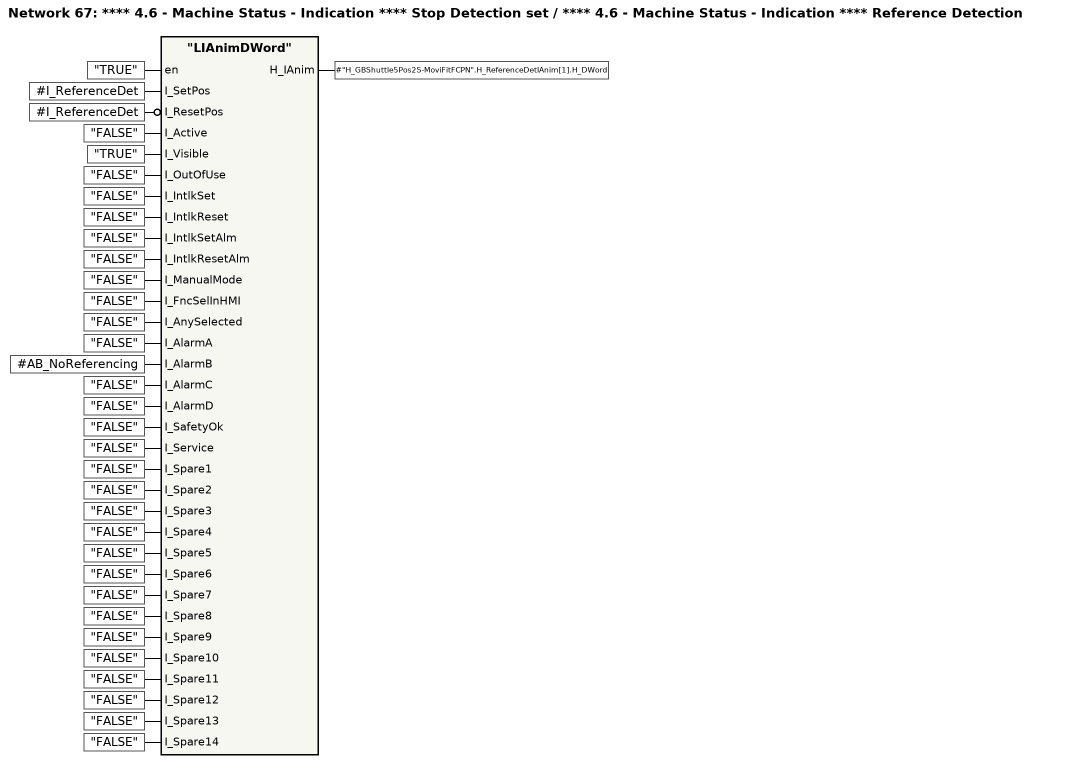
   IF "TRUE" THEN
       "LIAnimDWord"(I_SetPos := #I_ReferenceDet,
                     I_ResetPos := NOT #I_ReferenceDet,
                     I_Active := "FALSE",
                     I_Visible := "TRUE",
                     I_OutOfUse := "FALSE",
                     I_IntlkSet := "FALSE",
                     I_IntlkReset := "FALSE",
                     I_IntlkSetAlm := "FALSE",
                     I_IntlkResetAlm := "FALSE",
                     I_ManualMode := "FALSE",
                     I_FncSelInHMI := "FALSE",
                     I_AnySelected := "FALSE",
                     I_AlarmA := "FALSE",
                     I_AlarmB := #AB_NoReferencing,
                     I_AlarmC := "FALSE",
                     I_AlarmD := "FALSE",
                     I_SafetyOk := "FALSE",
                     I_Service := "FALSE",
                     I_Spare1 := "FALSE",
                     I_Spare2 := "FALSE",
                     I_Spare3 := "FALSE",
                     I_Spare4 := "FALSE",
                     I_Spare5 := "FALSE",
                     I_Spare6 := "FALSE",
                     I_Spare7 := "FALSE",
                     I_Spare8 := "FALSE",
                     I_Spare9 := "FALSE",
                     I_Spare10 := "FALSE",
                     I_Spare11 := "FALSE",
                     I_Spare12 := "FALSE",
                     I_Spare13 := "FALSE",
                     I_Spare14 := "FALSE",
                     H_IAnim => #"H_GBShuttle5Pos2S-MoviFitFCPN".H_ReferenceDetIAnim[1].H_DWord);
   END_IF;
END_REGION

REGION Network 68: **** 4.6 - Machine status - Indications **** Icon Animation
   // Animation for HMI
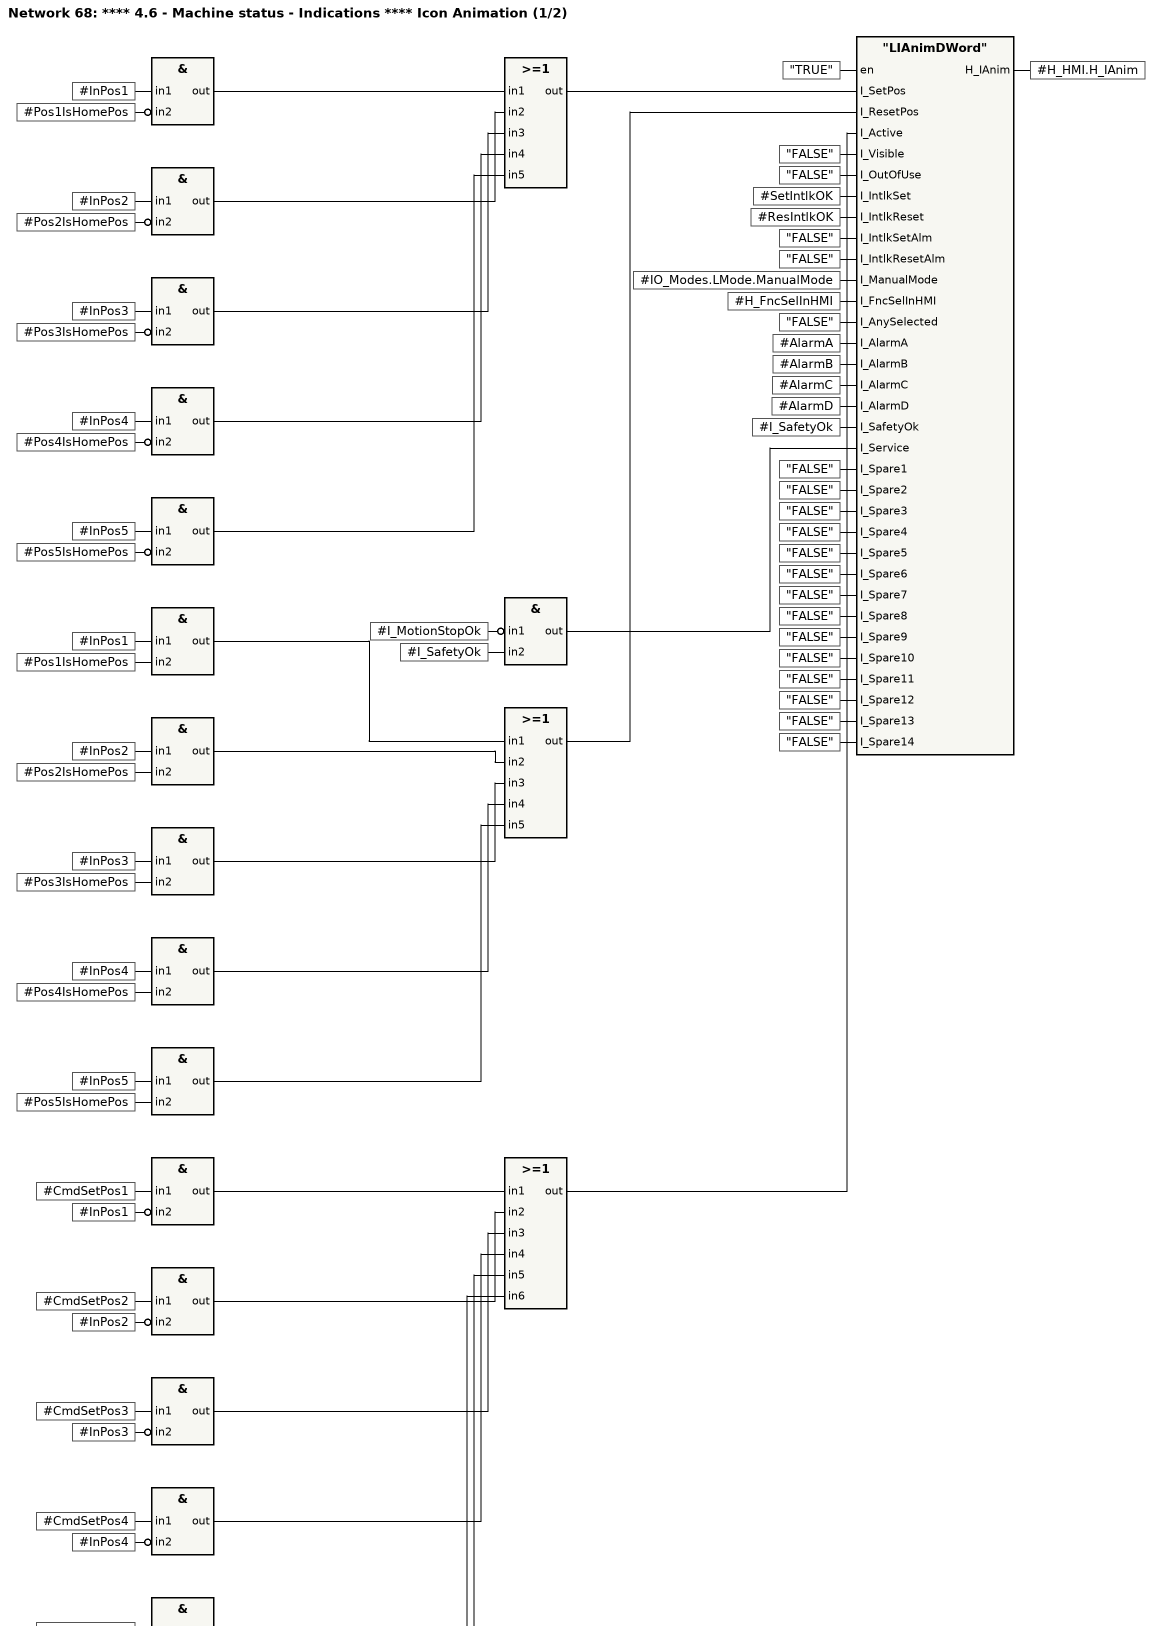
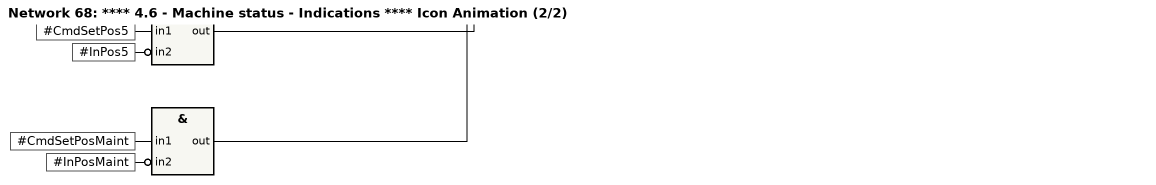
   IF "TRUE" THEN
       "LIAnimDWord"(I_SetPos := (#InPos1 AND NOT #Pos1IsHomePos) OR (#InPos2 AND NOT #Pos2IsHomePos) OR (#InPos3 AND NOT #Pos3IsHomePos) OR (#InPos4 AND NOT #Pos4IsHomePos) OR (#InPos5 AND NOT #Pos5IsHomePos),
                     I_ResetPos := (#InPos1 AND #Pos1IsHomePos) OR (#InPos2 AND #Pos2IsHomePos) OR (#InPos3 AND #Pos3IsHomePos) OR (#InPos4 AND #Pos4IsHomePos) OR (#InPos5 AND #Pos5IsHomePos),
                     I_Active := (#CmdSetPos1 AND NOT #InPos1) OR (#CmdSetPos2 AND NOT #InPos2) OR (#CmdSetPos3 AND NOT #InPos3) OR (#CmdSetPos4 AND NOT #InPos4) OR (#CmdSetPos5 AND NOT #InPos5) OR (#CmdSetPosMaint AND NOT #InPosMaint),
                     I_Visible := "FALSE",
                     I_OutOfUse := "FALSE",
                     I_IntlkSet := #SetIntlkOK,
                     I_IntlkReset := #ResIntlkOK,
                     I_IntlkSetAlm := "FALSE",
                     I_IntlkResetAlm := "FALSE",
                     I_ManualMode := #IO_Modes.LMode.ManualMode,
                     I_FncSelInHMI := #H_FncSelInHMI,
                     I_AnySelected := "FALSE",
                     I_AlarmA := #AlarmA,
                     I_AlarmB := #AlarmB,
                     I_AlarmC := #AlarmC,
                     I_AlarmD := #AlarmD,
                     I_SafetyOk := #I_SafetyOk,
                     I_Service := NOT #I_MotionStopOk AND #I_SafetyOk,
                     I_Spare1 := "FALSE",
                     I_Spare2 := "FALSE",
                     I_Spare3 := "FALSE",
                     I_Spare4 := "FALSE",
                     I_Spare5 := "FALSE",
                     I_Spare6 := "FALSE",
                     I_Spare7 := "FALSE",
                     I_Spare8 := "FALSE",
                     I_Spare9 := "FALSE",
                     I_Spare10 := "FALSE",
                     I_Spare11 := "FALSE",
                     I_Spare12 := "FALSE",
                     I_Spare13 := "FALSE",
                     I_Spare14 := "FALSE",
                     H_IAnim => #H_HMI.H_IAnim);
   END_IF;
END_REGION

REGION Network 69: **** 4.6 - Machine status - Indications **** Anim / **** 4.6 - Machine status - Indications **** Animation
   // Animation for HMI
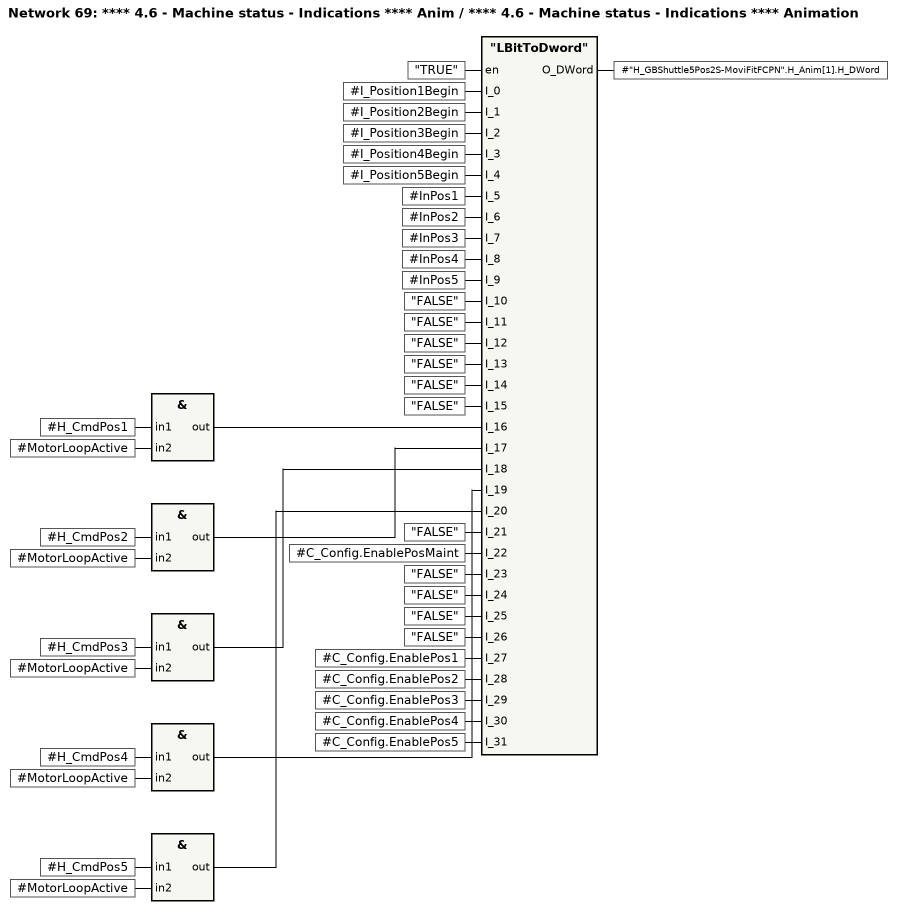
   IF "TRUE" THEN
       "LBitToDword"(I_0 := #I_Position1Begin,
                     I_1 := #I_Position2Begin,
                     I_2 := #I_Position3Begin,
                     I_3 := #I_Position4Begin,
                     I_4 := #I_Position5Begin,
                     I_5 := #InPos1,
                     I_6 := #InPos2,
                     I_7 := #InPos3,
                     I_8 := #InPos4,
                     I_9 := #InPos5,
                     I_10 := "FALSE",
                     I_11 := "FALSE",
                     I_12 := "FALSE",
                     I_13 := "FALSE",
                     I_14 := "FALSE",
                     I_15 := "FALSE",
                     I_16 := #H_CmdPos1 AND #MotorLoopActive,
                     I_17 := #H_CmdPos2 AND #MotorLoopActive,
                     I_18 := #H_CmdPos3 AND #MotorLoopActive,
                     I_19 := #H_CmdPos4 AND #MotorLoopActive,
                     I_20 := #H_CmdPos5 AND #MotorLoopActive,
                     I_21 := "FALSE",
                     I_22 := #C_Config.EnablePosMaint,
                     I_23 := "FALSE",
                     I_24 := "FALSE",
                     I_25 := "FALSE",
                     I_26 := "FALSE",
                     I_27 := #C_Config.EnablePos1,
                     I_28 := #C_Config.EnablePos2,
                     I_29 := #C_Config.EnablePos3,
                     I_30 := #C_Config.EnablePos4,
                     I_31 := #C_Config.EnablePos5,
                     O_DWord => #"H_GBShuttle5Pos2S-MoviFitFCPN".H_Anim[1].H_DWord);
   END_IF;
END_REGION

REGION Network 70: **** 4.6 - Machine status - Indications **** Anim / **** 4.6 - Machine status - Indications **** Animation
   // Animation for HMI
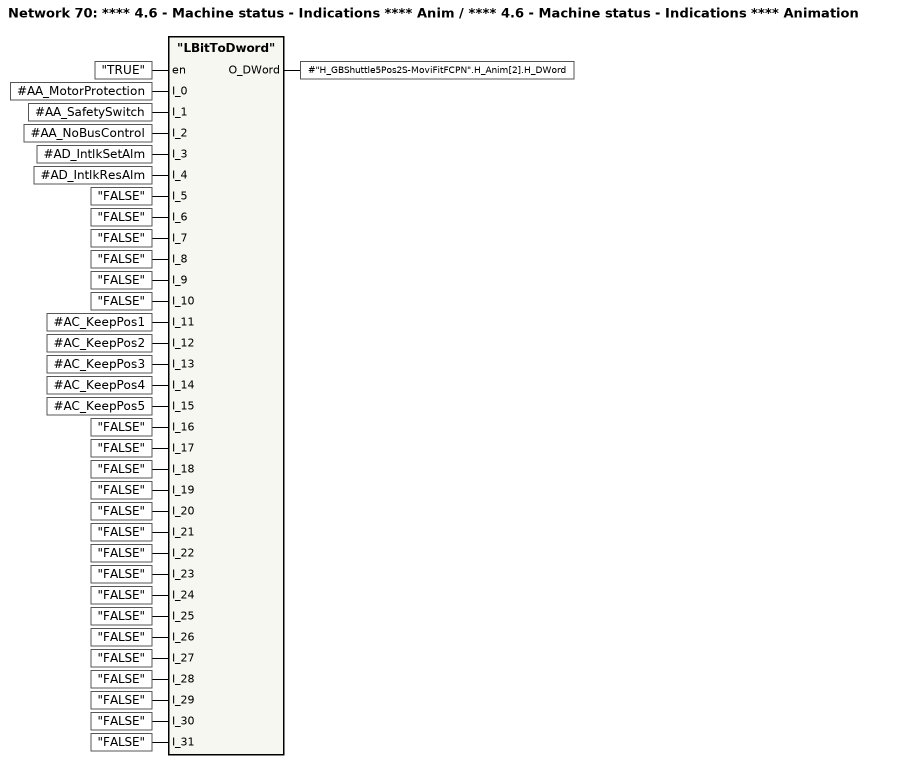
   IF "TRUE" THEN
       "LBitToDword"(I_0 := #AA_MotorProtection,
                     I_1 := #AA_SafetySwitch,
                     I_2 := #AA_NoBusControl,
                     I_3 := #AD_IntlkSetAlm,
                     I_4 := #AD_IntlkResAlm,
                     I_5 := "FALSE",
                     I_6 := "FALSE",
                     I_7 := "FALSE",
                     I_8 := "FALSE",
                     I_9 := "FALSE",
                     I_10 := "FALSE",
                     I_11 := #AC_KeepPos1,
                     I_12 := #AC_KeepPos2,
                     I_13 := #AC_KeepPos3,
                     I_14 := #AC_KeepPos4,
                     I_15 := #AC_KeepPos5,
                     I_16 := "FALSE",
                     I_17 := "FALSE",
                     I_18 := "FALSE",
                     I_19 := "FALSE",
                     I_20 := "FALSE",
                     I_21 := "FALSE",
                     I_22 := "FALSE",
                     I_23 := "FALSE",
                     I_24 := "FALSE",
                     I_25 := "FALSE",
                     I_26 := "FALSE",
                     I_27 := "FALSE",
                     I_28 := "FALSE",
                     I_29 := "FALSE",
                     I_30 := "FALSE",
                     I_31 := "FALSE",
                     O_DWord => #"H_GBShuttle5Pos2S-MoviFitFCPN".H_Anim[2].H_DWord);
   END_IF;
END_REGION

REGION Network 71: **** 4.6 - Machine status - Indications **** Anim / **** 4.6 - Machine status - Indications **** Animation
   // Animation for HMI
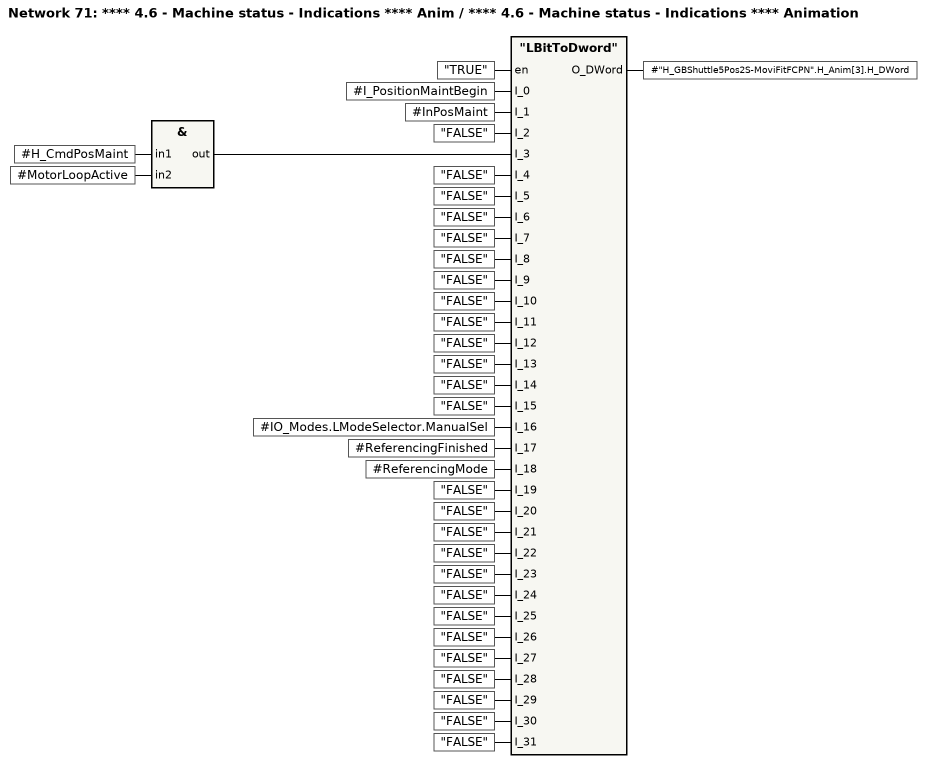
   IF "TRUE" THEN
       "LBitToDword"(I_0 := #I_PositionMaintBegin,
                     I_1 := #InPosMaint,
                     I_2 := "FALSE",
                     I_3 := #H_CmdPosMaint AND #MotorLoopActive,
                     I_4 := "FALSE",
                     I_5 := "FALSE",
                     I_6 := "FALSE",
                     I_7 := "FALSE",
                     I_8 := "FALSE",
                     I_9 := "FALSE",
                     I_10 := "FALSE",
                     I_11 := "FALSE",
                     I_12 := "FALSE",
                     I_13 := "FALSE",
                     I_14 := "FALSE",
                     I_15 := "FALSE",
                     I_16 := #IO_Modes.LModeSelector.ManualSel,
                     I_17 := #ReferencingFinished,
                     I_18 := #ReferencingMode,
                     I_19 := "FALSE",
                     I_20 := "FALSE",
                     I_21 := "FALSE",
                     I_22 := "FALSE",
                     I_23 := "FALSE",
                     I_24 := "FALSE",
                     I_25 := "FALSE",
                     I_26 := "FALSE",
                     I_27 := "FALSE",
                     I_28 := "FALSE",
                     I_29 := "FALSE",
                     I_30 := "FALSE",
                     I_31 := "FALSE",
                     O_DWord => #"H_GBShuttle5Pos2S-MoviFitFCPN".H_Anim[3].H_DWord);
   END_IF;
END_REGION

REGION Network 72: **** 4.6 - Machine status - Indications **** Anim / **** 4.6 - Machine status - Indications **** Animation
   // Anim
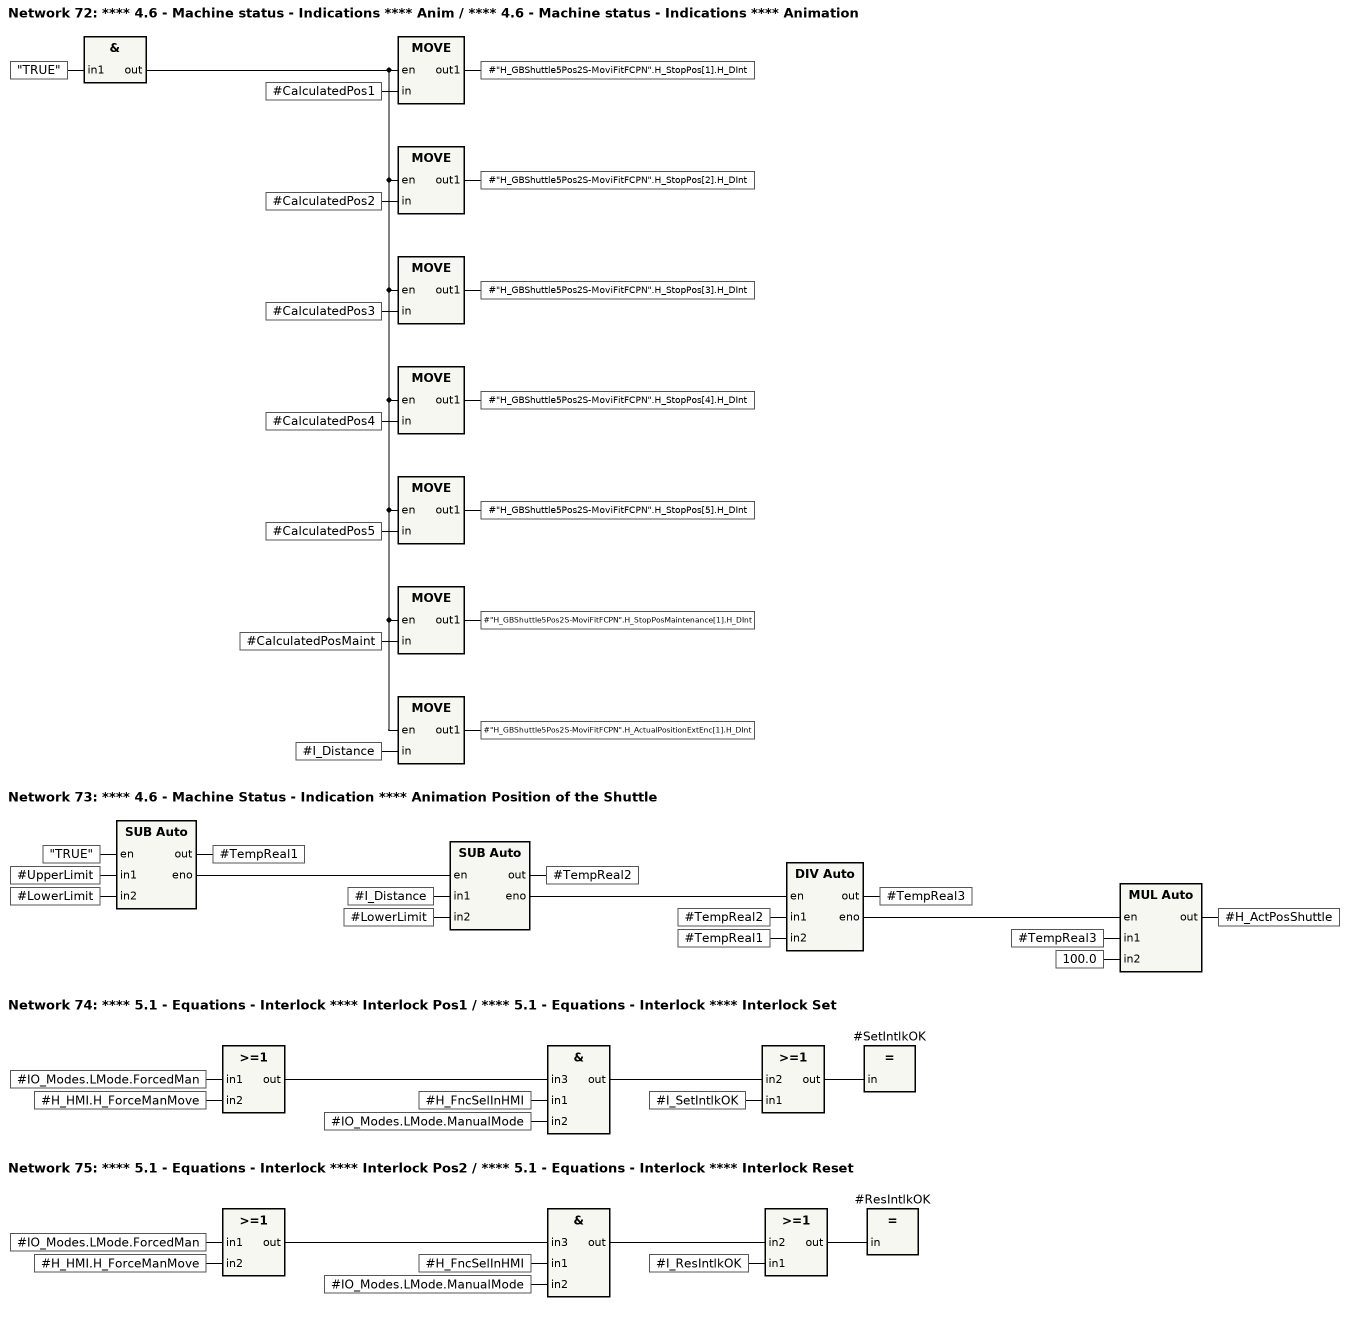
   IF "TRUE" THEN
       #"H_GBShuttle5Pos2S-MoviFitFCPN".H_StopPos[1].H_DInt := #CalculatedPos1;
       #"H_GBShuttle5Pos2S-MoviFitFCPN".H_StopPos[2].H_DInt := #CalculatedPos2;
       #"H_GBShuttle5Pos2S-MoviFitFCPN".H_StopPos[3].H_DInt := #CalculatedPos3;
       #"H_GBShuttle5Pos2S-MoviFitFCPN".H_StopPos[4].H_DInt := #CalculatedPos4;
       #"H_GBShuttle5Pos2S-MoviFitFCPN".H_StopPos[5].H_DInt := #CalculatedPos5;
       #"H_GBShuttle5Pos2S-MoviFitFCPN".H_StopPosMaintenance[1].H_DInt := #CalculatedPosMaint;
       #"H_GBShuttle5Pos2S-MoviFitFCPN".H_ActualPositionExtEnc[1].H_DInt := #I_Distance;
   END_IF;
END_REGION

REGION Network 73: **** 4.6 - Machine Status - Indication **** Animation Position of the Shuttle
   IF "TRUE" THEN
       #TempReal1 := #UpperLimit - #LowerLimit;
       #TempReal2 := #I_Distance - #LowerLimit;
       #TempReal3 := #TempReal2 / #TempReal1;
       #H_ActPosShuttle := #TempReal3 * 100.0;
   END_IF;
END_REGION

REGION Network 74: **** 5.1 - Equations - Interlock **** Interlock Pos1 / **** 5.1 - Equations - Interlock **** Interlock Set
   // Interlock
   #SetIntlkOK := ((#IO_Modes.LMode.ForcedMan OR #H_HMI.H_ForceManMove) AND #H_FncSelInHMI AND #IO_Modes.LMode.ManualMode) OR #I_SetIntlkOK;
END_REGION

REGION Network 75: **** 5.1 - Equations - Interlock **** Interlock Pos2 / **** 5.1 - Equations - Interlock **** Interlock Reset
   // Interlock
   #ResIntlkOK := ((#IO_Modes.LMode.ForcedMan OR #H_HMI.H_ForceManMove) AND #H_FncSelInHMI AND #IO_Modes.LMode.ManualMode) OR #I_ResIntlkOK;
END_REGION

REGION Network 76: **** 5.2 - Equations - Equations **** Alarm Condition Keep Position 1
   // Alarm Condition Keep Position
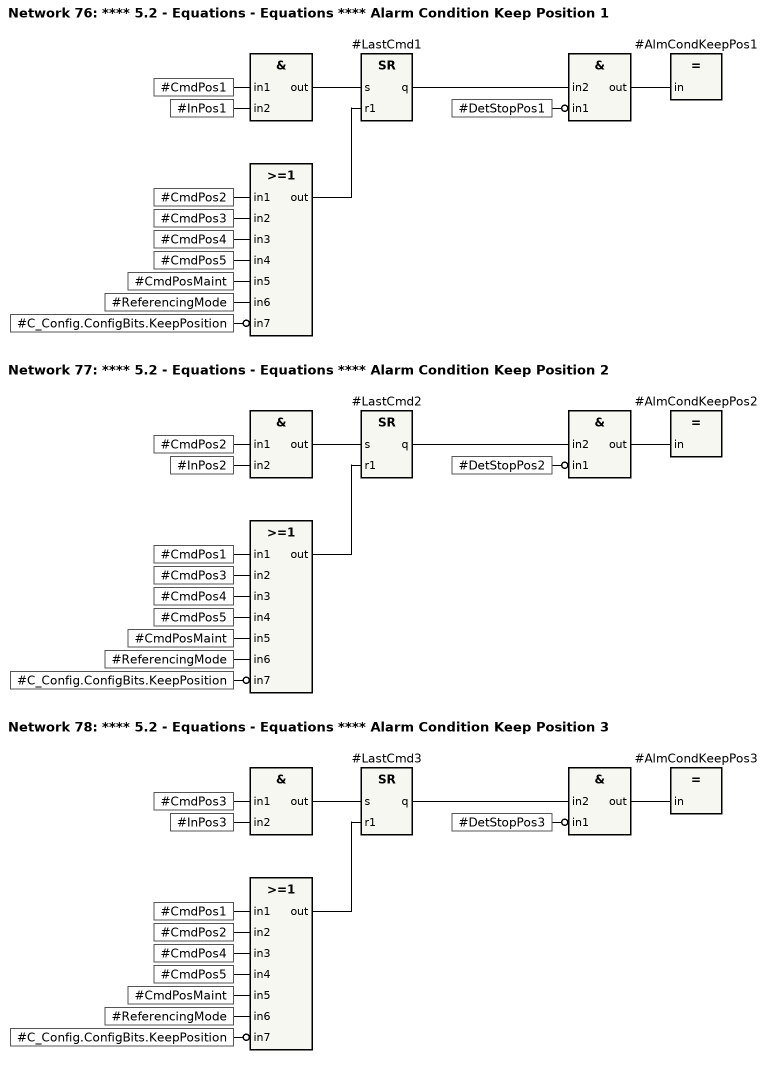
   IF #CmdPos1 AND #InPos1 THEN
       #LastCmd1 := TRUE;   // SR flip-flop
   END_IF;
   IF #CmdPos2 OR #CmdPos3 OR #CmdPos4 OR #CmdPos5 OR #CmdPosMaint OR #ReferencingMode OR NOT #C_Config.ConfigBits.KeepPosition THEN
       #LastCmd1 := FALSE;
   END_IF;
   #AlmCondKeepPos1 := #LastCmd1 AND NOT #DetStopPos1;
END_REGION

REGION Network 77: **** 5.2 - Equations - Equations **** Alarm Condition Keep Position 2
   // Alarm Condition Keep Position
   IF #CmdPos2 AND #InPos2 THEN
       #LastCmd2 := TRUE;   // SR flip-flop
   END_IF;
   IF #CmdPos1 OR #CmdPos3 OR #CmdPos4 OR #CmdPos5 OR #CmdPosMaint OR #ReferencingMode OR NOT #C_Config.ConfigBits.KeepPosition THEN
       #LastCmd2 := FALSE;
   END_IF;
   #AlmCondKeepPos2 := #LastCmd2 AND NOT #DetStopPos2;
END_REGION

REGION Network 78: **** 5.2 - Equations - Equations **** Alarm Condition Keep Position 3
   // Alarm Condition Keep Position
   IF #CmdPos3 AND #InPos3 THEN
       #LastCmd3 := TRUE;   // SR flip-flop
   END_IF;
   IF #CmdPos1 OR #CmdPos2 OR #CmdPos4 OR #CmdPos5 OR #CmdPosMaint OR #ReferencingMode OR NOT #C_Config.ConfigBits.KeepPosition THEN
       #LastCmd3 := FALSE;
   END_IF;
   #AlmCondKeepPos3 := #LastCmd3 AND NOT #DetStopPos3;
END_REGION

REGION Network 79: **** 5.2 - Equations - Equations **** Alarm Condition Keep Position 4
   // Alarm Condition Keep Position
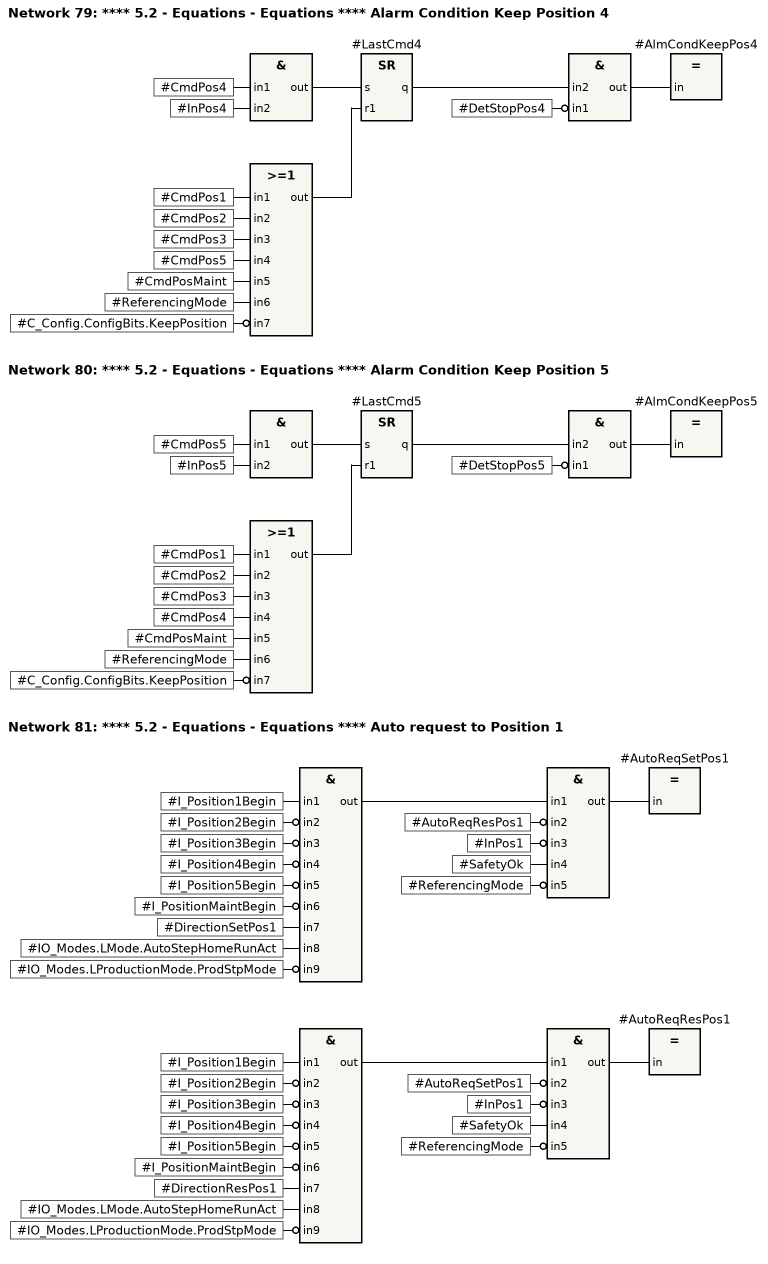
   IF #CmdPos4 AND #InPos4 THEN
       #LastCmd4 := TRUE;   // SR flip-flop
   END_IF;
   IF #CmdPos1 OR #CmdPos2 OR #CmdPos3 OR #CmdPos5 OR #CmdPosMaint OR #ReferencingMode OR NOT #C_Config.ConfigBits.KeepPosition THEN
       #LastCmd4 := FALSE;
   END_IF;
   #AlmCondKeepPos4 := #LastCmd4 AND NOT #DetStopPos4;
END_REGION

REGION Network 80: **** 5.2 - Equations - Equations **** Alarm Condition Keep Position 5
   // Alarm Condition Keep Position
   IF #CmdPos5 AND #InPos5 THEN
       #LastCmd5 := TRUE;   // SR flip-flop
   END_IF;
   IF #CmdPos1 OR #CmdPos2 OR #CmdPos3 OR #CmdPos4 OR #CmdPosMaint OR #ReferencingMode OR NOT #C_Config.ConfigBits.KeepPosition THEN
       #LastCmd5 := FALSE;
   END_IF;
   #AlmCondKeepPos5 := #LastCmd5 AND NOT #DetStopPos5;
END_REGION

REGION Network 81: **** 5.2 - Equations - Equations **** Auto request to Position 1
   // AutoReq Pos 1
   #AutoReqSetPos1 := #I_Position1Begin AND NOT #I_Position2Begin AND NOT #I_Position3Begin AND NOT #I_Position4Begin AND NOT #I_Position5Begin AND NOT #I_PositionMaintBegin AND #DirectionSetPos1 AND #IO_Modes.LMode.AutoStepHomeRunAct AND NOT #IO_Modes.LProductionMode.ProdStpMode AND NOT #AutoReqResPos1 AND NOT #InPos1 AND #SafetyOk AND NOT #ReferencingMode;
   #AutoReqResPos1 := #I_Position1Begin AND NOT #I_Position2Begin AND NOT #I_Position3Begin AND NOT #I_Position4Begin AND NOT #I_Position5Begin AND NOT #I_PositionMaintBegin AND #DirectionResPos1 AND #IO_Modes.LMode.AutoStepHomeRunAct AND NOT #IO_Modes.LProductionMode.ProdStpMode AND NOT #AutoReqSetPos1 AND NOT #InPos1 AND #SafetyOk AND NOT #ReferencingMode;
END_REGION

REGION Network 82: **** 5.2 - Equations - Equations **** Auto request to Position 2
   // AutoReq Pos 1
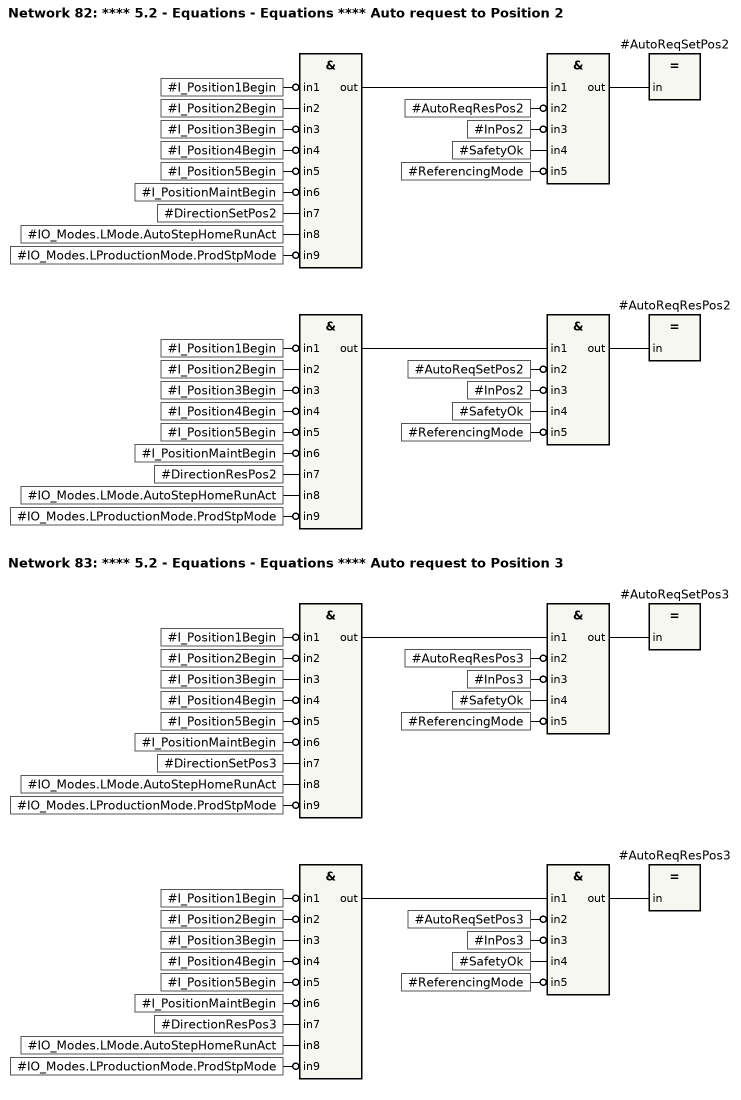
   #AutoReqSetPos2 := NOT #I_Position1Begin AND #I_Position2Begin AND NOT #I_Position3Begin AND NOT #I_Position4Begin AND NOT #I_Position5Begin AND NOT #I_PositionMaintBegin AND #DirectionSetPos2 AND #IO_Modes.LMode.AutoStepHomeRunAct AND NOT #IO_Modes.LProductionMode.ProdStpMode AND NOT #AutoReqResPos2 AND NOT #InPos2 AND #SafetyOk AND NOT #ReferencingMode;
   #AutoReqResPos2 := NOT #I_Position1Begin AND #I_Position2Begin AND NOT #I_Position3Begin AND NOT #I_Position4Begin AND NOT #I_Position5Begin AND NOT #I_PositionMaintBegin AND #DirectionResPos2 AND #IO_Modes.LMode.AutoStepHomeRunAct AND NOT #IO_Modes.LProductionMode.ProdStpMode AND NOT #AutoReqSetPos2 AND NOT #InPos2 AND #SafetyOk AND NOT #ReferencingMode;
END_REGION

REGION Network 83: **** 5.2 - Equations - Equations **** Auto request to Position 3
   // AutoReq Pos 1
   #AutoReqSetPos3 := NOT #I_Position1Begin AND NOT #I_Position2Begin AND #I_Position3Begin AND NOT #I_Position4Begin AND NOT #I_Position5Begin AND NOT #I_PositionMaintBegin AND #DirectionSetPos3 AND #IO_Modes.LMode.AutoStepHomeRunAct AND NOT #IO_Modes.LProductionMode.ProdStpMode AND NOT #AutoReqResPos3 AND NOT #InPos3 AND #SafetyOk AND NOT #ReferencingMode;
   #AutoReqResPos3 := NOT #I_Position1Begin AND NOT #I_Position2Begin AND #I_Position3Begin AND NOT #I_Position4Begin AND NOT #I_Position5Begin AND NOT #I_PositionMaintBegin AND #DirectionResPos3 AND #IO_Modes.LMode.AutoStepHomeRunAct AND NOT #IO_Modes.LProductionMode.ProdStpMode AND NOT #AutoReqSetPos3 AND NOT #InPos3 AND #SafetyOk AND NOT #ReferencingMode;
END_REGION

REGION Network 84: **** 5.2 - Equations - Equations **** Auto request to Position 4
   // AutoReq Pos 1
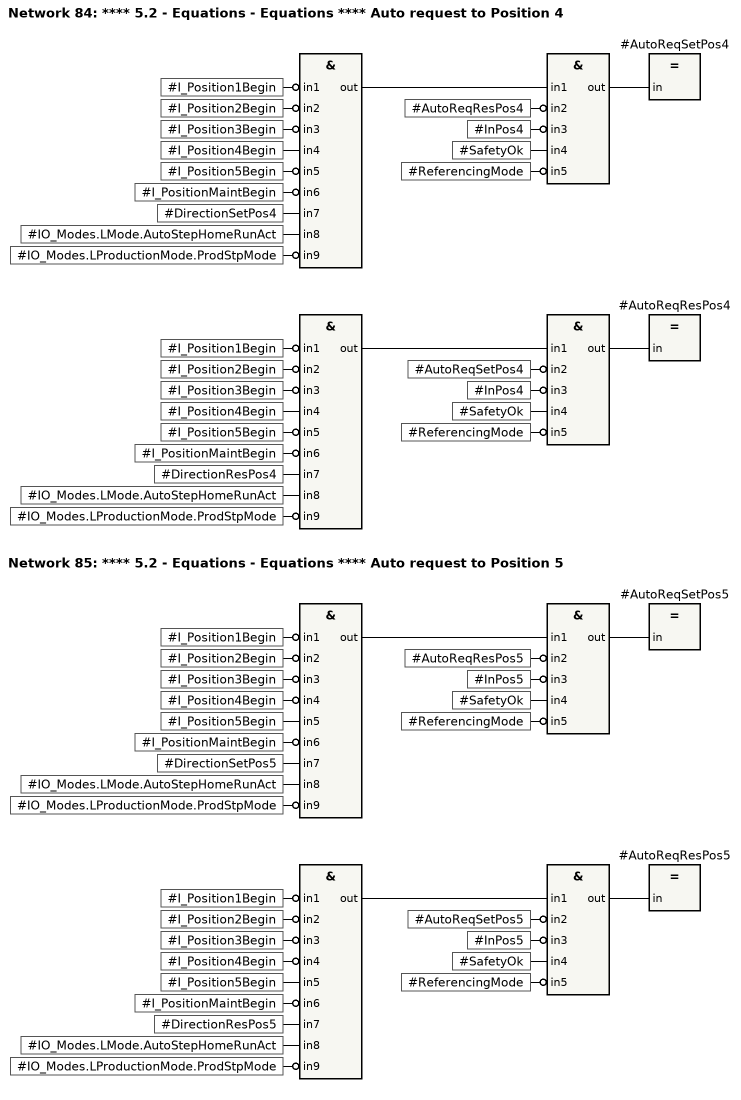
   #AutoReqSetPos4 := NOT #I_Position1Begin AND NOT #I_Position2Begin AND NOT #I_Position3Begin AND #I_Position4Begin AND NOT #I_Position5Begin AND NOT #I_PositionMaintBegin AND #DirectionSetPos4 AND #IO_Modes.LMode.AutoStepHomeRunAct AND NOT #IO_Modes.LProductionMode.ProdStpMode AND NOT #AutoReqResPos4 AND NOT #InPos4 AND #SafetyOk AND NOT #ReferencingMode;
   #AutoReqResPos4 := NOT #I_Position1Begin AND NOT #I_Position2Begin AND NOT #I_Position3Begin AND #I_Position4Begin AND NOT #I_Position5Begin AND NOT #I_PositionMaintBegin AND #DirectionResPos4 AND #IO_Modes.LMode.AutoStepHomeRunAct AND NOT #IO_Modes.LProductionMode.ProdStpMode AND NOT #AutoReqSetPos4 AND NOT #InPos4 AND #SafetyOk AND NOT #ReferencingMode;
END_REGION

REGION Network 85: **** 5.2 - Equations - Equations **** Auto request to Position 5
   // AutoReq Pos 1
   #AutoReqSetPos5 := NOT #I_Position1Begin AND NOT #I_Position2Begin AND NOT #I_Position3Begin AND NOT #I_Position4Begin AND #I_Position5Begin AND NOT #I_PositionMaintBegin AND #DirectionSetPos5 AND #IO_Modes.LMode.AutoStepHomeRunAct AND NOT #IO_Modes.LProductionMode.ProdStpMode AND NOT #AutoReqResPos5 AND NOT #InPos5 AND #SafetyOk AND NOT #ReferencingMode;
   #AutoReqResPos5 := NOT #I_Position1Begin AND NOT #I_Position2Begin AND NOT #I_Position3Begin AND NOT #I_Position4Begin AND #I_Position5Begin AND NOT #I_PositionMaintBegin AND #DirectionResPos5 AND #IO_Modes.LMode.AutoStepHomeRunAct AND NOT #IO_Modes.LProductionMode.ProdStpMode AND NOT #AutoReqSetPos5 AND NOT #InPos5 AND #SafetyOk AND NOT #ReferencingMode;
END_REGION

REGION Network 86: **** 5.2 - Equations - Equations **** Auto request to Position Maintenance
   // AutoReq Pos 1
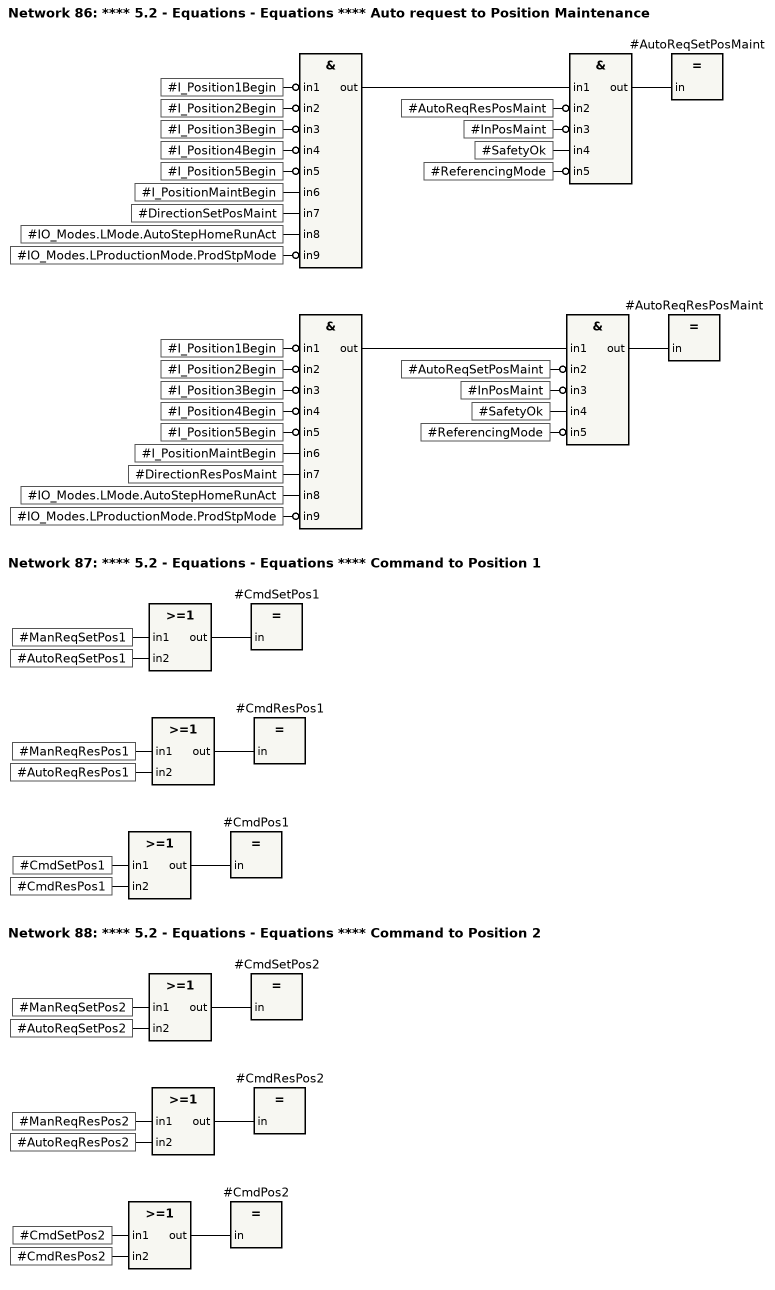
   #AutoReqSetPosMaint := NOT #I_Position1Begin AND NOT #I_Position2Begin AND NOT #I_Position3Begin AND NOT #I_Position4Begin AND NOT #I_Position5Begin AND #I_PositionMaintBegin AND #DirectionSetPosMaint AND #IO_Modes.LMode.AutoStepHomeRunAct AND NOT #IO_Modes.LProductionMode.ProdStpMode AND NOT #AutoReqResPosMaint AND NOT #InPosMaint AND #SafetyOk AND NOT #ReferencingMode;
   #AutoReqResPosMaint := NOT #I_Position1Begin AND NOT #I_Position2Begin AND NOT #I_Position3Begin AND NOT #I_Position4Begin AND NOT #I_Position5Begin AND #I_PositionMaintBegin AND #DirectionResPosMaint AND #IO_Modes.LMode.AutoStepHomeRunAct AND NOT #IO_Modes.LProductionMode.ProdStpMode AND NOT #AutoReqSetPosMaint AND NOT #InPosMaint AND #SafetyOk AND NOT #ReferencingMode;
END_REGION

REGION Network 87: **** 5.2 - Equations - Equations **** Command to Position 1
   #CmdSetPos1 := #ManReqSetPos1 OR #AutoReqSetPos1;
   #CmdResPos1 := #ManReqResPos1 OR #AutoReqResPos1;
   #CmdPos1 := #CmdSetPos1 OR #CmdResPos1;
END_REGION

REGION Network 88: **** 5.2 - Equations - Equations **** Command to Position 2
   #CmdSetPos2 := #ManReqSetPos2 OR #AutoReqSetPos2;
   #CmdResPos2 := #ManReqResPos2 OR #AutoReqResPos2;
   #CmdPos2 := #CmdSetPos2 OR #CmdResPos2;
END_REGION

REGION Network 89: **** 5.2 - Equations - Equations **** Command to Position 3
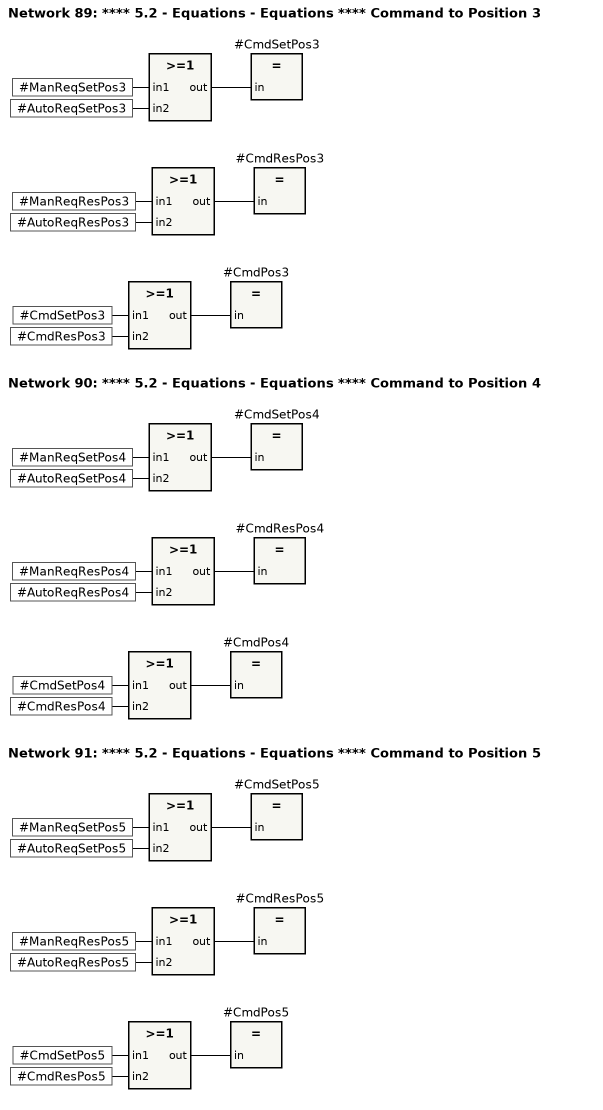
   #CmdSetPos3 := #ManReqSetPos3 OR #AutoReqSetPos3;
   #CmdResPos3 := #ManReqResPos3 OR #AutoReqResPos3;
   #CmdPos3 := #CmdSetPos3 OR #CmdResPos3;
END_REGION

REGION Network 90: **** 5.2 - Equations - Equations **** Command to Position 4
   #CmdSetPos4 := #ManReqSetPos4 OR #AutoReqSetPos4;
   #CmdResPos4 := #ManReqResPos4 OR #AutoReqResPos4;
   #CmdPos4 := #CmdSetPos4 OR #CmdResPos4;
END_REGION

REGION Network 91: **** 5.2 - Equations - Equations **** Command to Position 5
   #CmdSetPos5 := #ManReqSetPos5 OR #AutoReqSetPos5;
   #CmdResPos5 := #ManReqResPos5 OR #AutoReqResPos5;
   #CmdPos5 := #CmdSetPos5 OR #CmdResPos5;
END_REGION

REGION Network 92: **** 5.2 - Equations - Equations **** Command to Position Maintenance
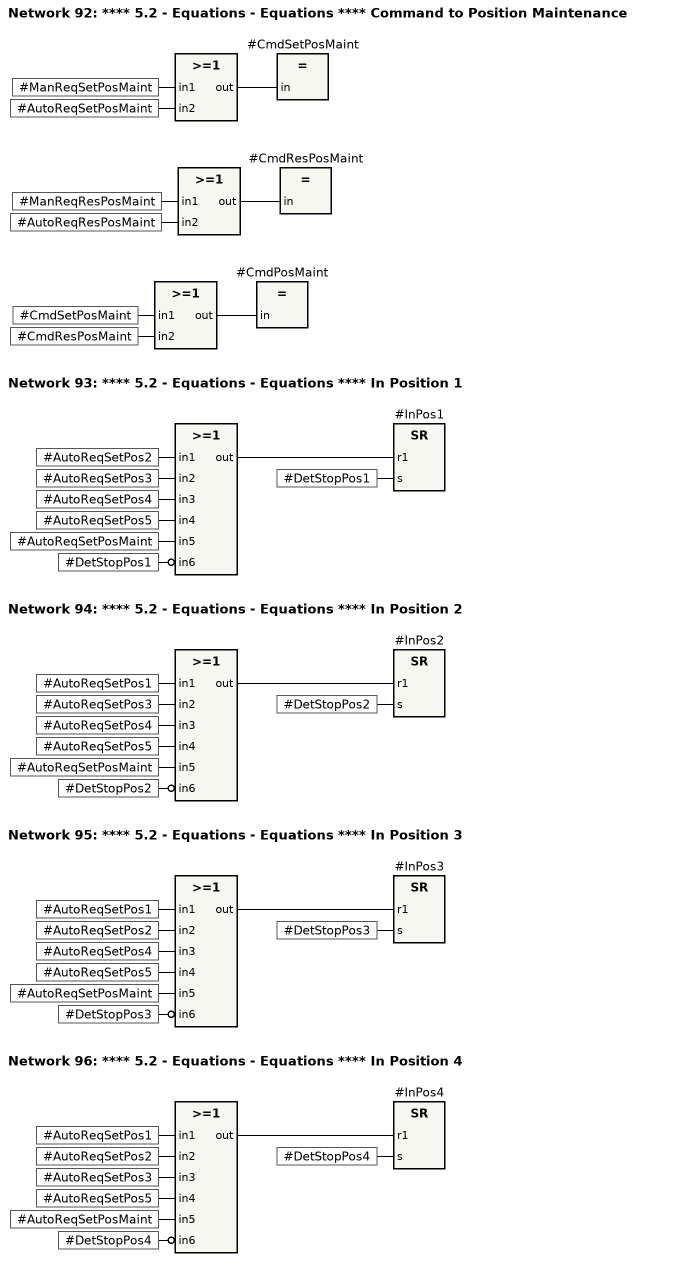
   #CmdSetPosMaint := #ManReqSetPosMaint OR #AutoReqSetPosMaint;
   #CmdResPosMaint := #ManReqResPosMaint OR #AutoReqResPosMaint;
   #CmdPosMaint := #CmdSetPosMaint OR #CmdResPosMaint;
END_REGION

REGION Network 93: **** 5.2 - Equations - Equations **** In Position 1
   IF #DetStopPos1 THEN
       #InPos1 := TRUE;   // SR flip-flop
   END_IF;
   IF #AutoReqSetPos2 OR #AutoReqSetPos3 OR #AutoReqSetPos4 OR #AutoReqSetPos5 OR #AutoReqSetPosMaint OR NOT #DetStopPos1 THEN
       #InPos1 := FALSE;
   END_IF;
END_REGION

REGION Network 94: **** 5.2 - Equations - Equations **** In Position 2
   IF #DetStopPos2 THEN
       #InPos2 := TRUE;   // SR flip-flop
   END_IF;
   IF #AutoReqSetPos1 OR #AutoReqSetPos3 OR #AutoReqSetPos4 OR #AutoReqSetPos5 OR #AutoReqSetPosMaint OR NOT #DetStopPos2 THEN
       #InPos2 := FALSE;
   END_IF;
END_REGION

REGION Network 95: **** 5.2 - Equations - Equations **** In Position 3
   IF #DetStopPos3 THEN
       #InPos3 := TRUE;   // SR flip-flop
   END_IF;
   IF #AutoReqSetPos1 OR #AutoReqSetPos2 OR #AutoReqSetPos4 OR #AutoReqSetPos5 OR #AutoReqSetPosMaint OR NOT #DetStopPos3 THEN
       #InPos3 := FALSE;
   END_IF;
END_REGION

REGION Network 96: **** 5.2 - Equations - Equations **** In Position 4
   IF #DetStopPos4 THEN
       #InPos4 := TRUE;   // SR flip-flop
   END_IF;
   IF #AutoReqSetPos1 OR #AutoReqSetPos2 OR #AutoReqSetPos3 OR #AutoReqSetPos5 OR #AutoReqSetPosMaint OR NOT #DetStopPos4 THEN
       #InPos4 := FALSE;
   END_IF;
END_REGION

REGION Network 97: **** 5.2 - Equations - Equations **** In Position 5
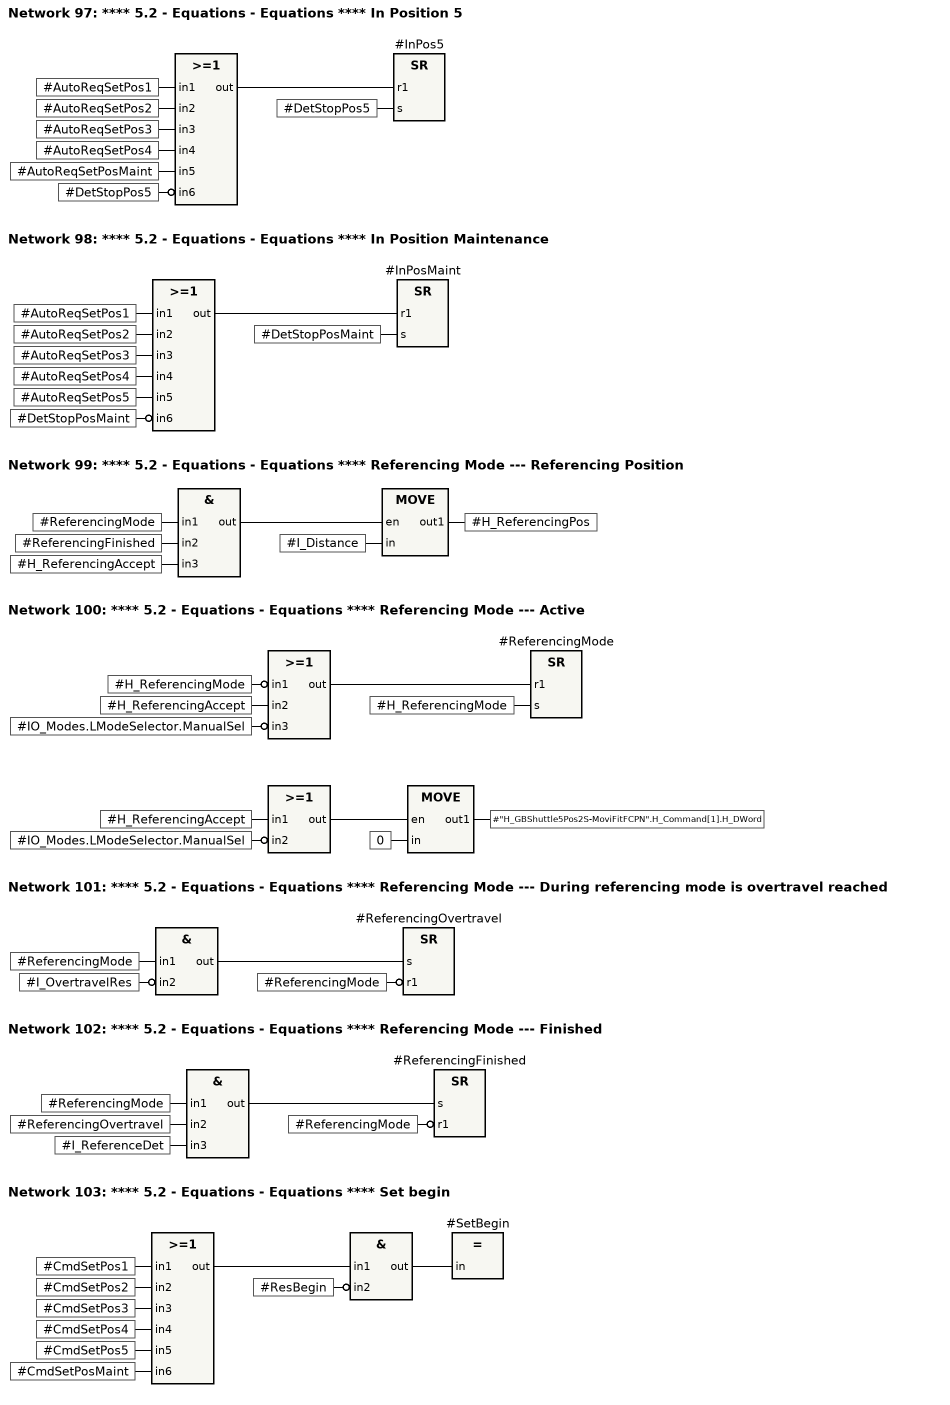
   IF #DetStopPos5 THEN
       #InPos5 := TRUE;   // SR flip-flop
   END_IF;
   IF #AutoReqSetPos1 OR #AutoReqSetPos2 OR #AutoReqSetPos3 OR #AutoReqSetPos4 OR #AutoReqSetPosMaint OR NOT #DetStopPos5 THEN
       #InPos5 := FALSE;
   END_IF;
END_REGION

REGION Network 98: **** 5.2 - Equations - Equations **** In Position Maintenance
   IF #DetStopPosMaint THEN
       #InPosMaint := TRUE;   // SR flip-flop
   END_IF;
   IF #AutoReqSetPos1 OR #AutoReqSetPos2 OR #AutoReqSetPos3 OR #AutoReqSetPos4 OR #AutoReqSetPos5 OR NOT #DetStopPosMaint THEN
       #InPosMaint := FALSE;
   END_IF;
END_REGION

REGION Network 99: **** 5.2 - Equations - Equations **** Referencing Mode --- Referencing Position
   IF #ReferencingMode AND #ReferencingFinished AND #H_ReferencingAccept THEN
       #H_ReferencingPos := #I_Distance;
   END_IF;
END_REGION

REGION Network 100: **** 5.2 - Equations - Equations **** Referencing Mode --- Active
   IF #H_ReferencingMode THEN
       #ReferencingMode := TRUE;   // SR flip-flop
   END_IF;
   IF NOT #H_ReferencingMode OR #H_ReferencingAccept OR NOT #IO_Modes.LModeSelector.ManualSel THEN
       #ReferencingMode := FALSE;
   END_IF;
   IF #H_ReferencingAccept OR NOT #IO_Modes.LModeSelector.ManualSel THEN
       #"H_GBShuttle5Pos2S-MoviFitFCPN".H_Command[1].H_DWord := 0;
   END_IF;
END_REGION

REGION Network 101: **** 5.2 - Equations - Equations **** Referencing Mode --- During referencing mode is overtravel reached
   IF #ReferencingMode AND NOT #I_OvertravelRes THEN
       #ReferencingOvertravel := TRUE;   // SR flip-flop
   END_IF;
   IF NOT #ReferencingMode THEN #ReferencingOvertravel := FALSE; END_IF;
END_REGION

REGION Network 102: **** 5.2 - Equations - Equations **** Referencing Mode --- Finished
   IF #ReferencingMode AND #ReferencingOvertravel AND #I_ReferenceDet THEN
       #ReferencingFinished := TRUE;   // SR flip-flop
   END_IF;
   IF NOT #ReferencingMode THEN #ReferencingFinished := FALSE; END_IF;
END_REGION

REGION Network 103: **** 5.2 - Equations - Equations **** Set begin
   #SetBegin := (#CmdSetPos1 OR #CmdSetPos2 OR #CmdSetPos3 OR #CmdSetPos4 OR #CmdSetPos5 OR #CmdSetPosMaint) AND NOT #ResBegin;
END_REGION

REGION Network 104: **** 5.2 - Equations - Equations **** Reset begin
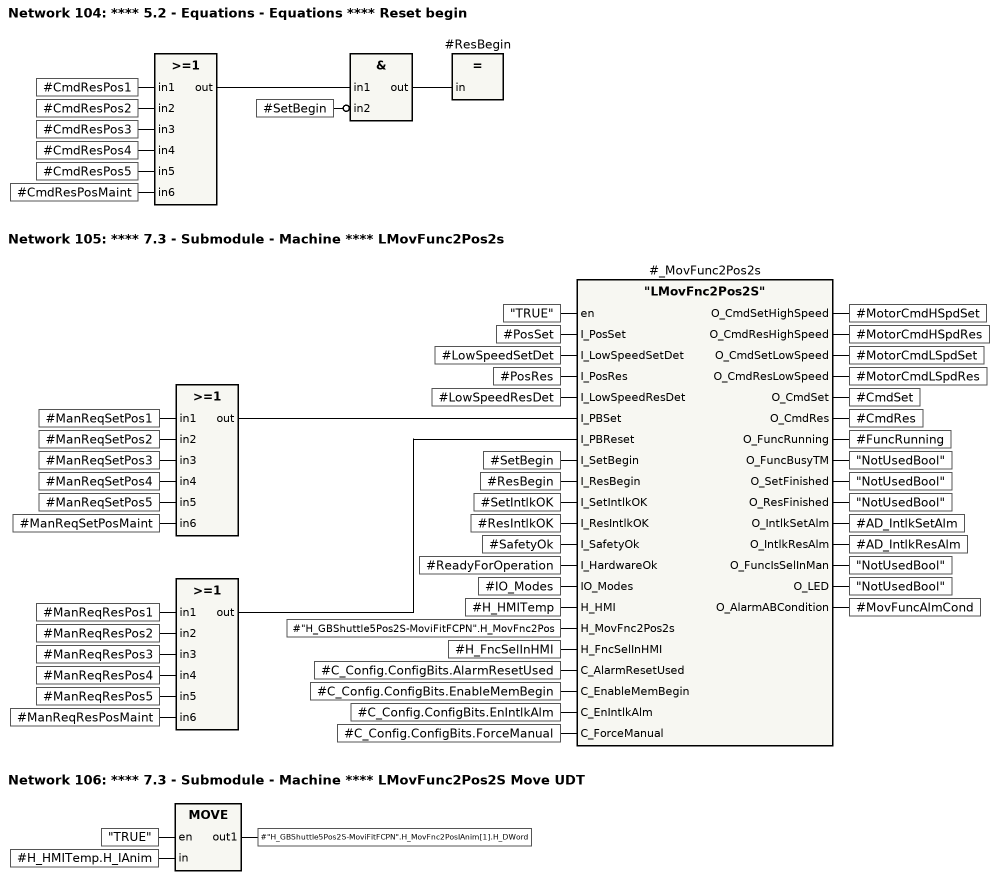
   #ResBegin := (#CmdResPos1 OR #CmdResPos2 OR #CmdResPos3 OR #CmdResPos4 OR #CmdResPos5 OR #CmdResPosMaint) AND NOT #SetBegin;
END_REGION

REGION Network 105: **** 7.3 - Submodule - Machine **** LMovFunc2Pos2s
   // LMovFunc2Pos
   IF "TRUE" THEN
       #_MovFunc2Pos2s(I_PosSet := #PosSet,   // "LMovFnc2Pos2S"
                       I_LowSpeedSetDet := #LowSpeedSetDet,
                       I_PosRes := #PosRes,
                       I_LowSpeedResDet := #LowSpeedResDet,
                       I_PBSet := #ManReqSetPos1 OR #ManReqSetPos2 OR #ManReqSetPos3 OR #ManReqSetPos4 OR #ManReqSetPos5 OR #ManReqSetPosMaint,
                       I_PBReset := #ManReqResPos1 OR #ManReqResPos2 OR #ManReqResPos3 OR #ManReqResPos4 OR #ManReqResPos5 OR #ManReqResPosMaint,
                       I_SetBegin := #SetBegin,
                       I_ResBegin := #ResBegin,
                       I_SetIntlkOK := #SetIntlkOK,
                       I_ResIntlkOK := #ResIntlkOK,
                       I_SafetyOk := #SafetyOk,
                       I_HardwareOk := #ReadyForOperation,
                       IO_Modes := #IO_Modes,
                       H_HMI := #H_HMITemp,
                       H_MovFnc2Pos2s := #"H_GBShuttle5Pos2S-MoviFitFCPN".H_MovFnc2Pos,
                       H_FncSelInHMI := #H_FncSelInHMI,
                       C_AlarmResetUsed := #C_Config.ConfigBits.AlarmResetUsed,
                       C_EnableMemBegin := #C_Config.ConfigBits.EnableMemBegin,
                       C_EnIntlkAlm := #C_Config.ConfigBits.EnIntlkAlm,
                       C_ForceManual := #C_Config.ConfigBits.ForceManual,
                       O_CmdSetHighSpeed => #MotorCmdHSpdSet,
                       O_CmdResHighSpeed => #MotorCmdHSpdRes,
                       O_CmdSetLowSpeed => #MotorCmdLSpdSet,
                       O_CmdResLowSpeed => #MotorCmdLSpdRes,
                       O_CmdSet => #CmdSet,
                       O_CmdRes => #CmdRes,
                       O_FuncRunning => #FuncRunning,
                       O_FuncBusyTM => "NotUsedBool",
                       O_SetFinished => "NotUsedBool",
                       O_ResFinished => "NotUsedBool",
                       O_IntlkSetAlm => #AD_IntlkSetAlm,
                       O_IntlkResAlm => #AD_IntlkResAlm,
                       O_FuncIsSelInMan => "NotUsedBool",
                       O_LED => "NotUsedBool",
                       O_AlarmABCondition => #MovFuncAlmCond);
   END_IF;
END_REGION

REGION Network 106: **** 7.3 - Submodule - Machine **** LMovFunc2Pos2S Move UDT
   // LMovFunc2Pos2S Move UDT
   IF "TRUE" THEN
       #"H_GBShuttle5Pos2S-MoviFitFCPN".H_MovFnc2PosIAnim[1].H_DWord := #H_HMITemp.H_IAnim;
   END_IF;
END_REGION

REGION Network 107: **** 7.3 - Submodule - Machine **** L2StopPos
   // L2StopPos
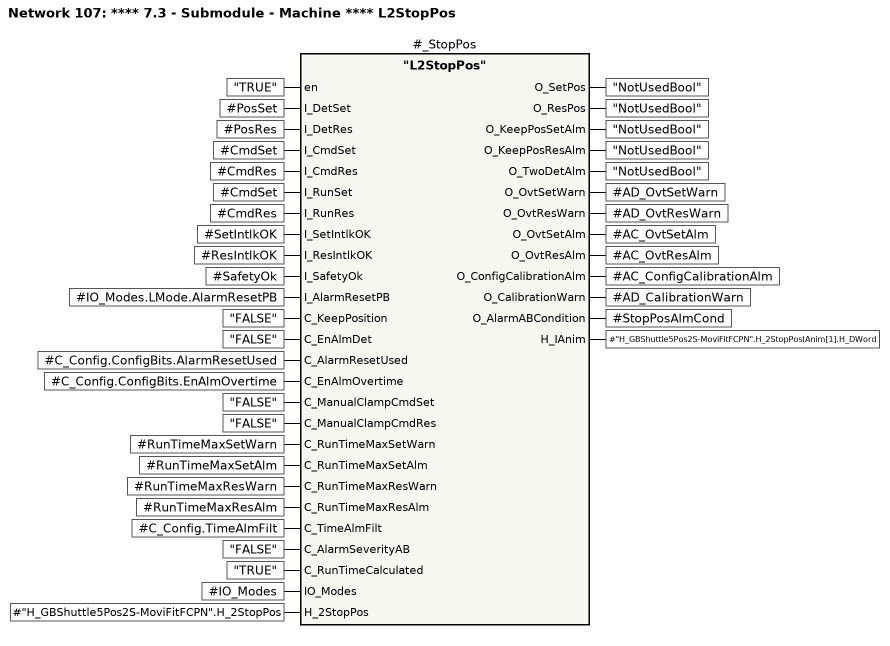
   IF "TRUE" THEN
       #_StopPos(I_DetSet := #PosSet,   // "L2StopPos"
                 I_DetRes := #PosRes,
                 I_CmdSet := #CmdSet,
                 I_CmdRes := #CmdRes,
                 I_RunSet := #CmdSet,
                 I_RunRes := #CmdRes,
                 I_SetIntlkOK := #SetIntlkOK,
                 I_ResIntlkOK := #ResIntlkOK,
                 I_SafetyOk := #SafetyOk,
                 I_AlarmResetPB := #IO_Modes.LMode.AlarmResetPB,
                 C_KeepPosition := "FALSE",
                 C_EnAlmDet := "FALSE",
                 C_AlarmResetUsed := #C_Config.ConfigBits.AlarmResetUsed,
                 C_EnAlmOvertime := #C_Config.ConfigBits.EnAlmOvertime,
                 C_ManualClampCmdSet := "FALSE",
                 C_ManualClampCmdRes := "FALSE",
                 C_RunTimeMaxSetWarn := #RunTimeMaxSetWarn,
                 C_RunTimeMaxSetAlm := #RunTimeMaxSetAlm,
                 C_RunTimeMaxResWarn := #RunTimeMaxResWarn,
                 C_RunTimeMaxResAlm := #RunTimeMaxResAlm,
                 C_TimeAlmFilt := #C_Config.TimeAlmFilt,
                 C_AlarmSeverityAB := "FALSE",
                 C_RunTimeCalculated := "TRUE",
                 IO_Modes := #IO_Modes,
                 H_2StopPos := #"H_GBShuttle5Pos2S-MoviFitFCPN".H_2StopPos,
                 O_SetPos => "NotUsedBool",
                 O_ResPos => "NotUsedBool",
                 O_KeepPosSetAlm => "NotUsedBool",
                 O_KeepPosResAlm => "NotUsedBool",
                 O_TwoDetAlm => "NotUsedBool",
                 O_OvtSetWarn => #AD_OvtSetWarn,
                 O_OvtResWarn => #AD_OvtResWarn,
                 O_OvtSetAlm => #AC_OvtSetAlm,
                 O_OvtResAlm => #AC_OvtResAlm,
                 O_ConfigCalibrationAlm => #AC_ConfigCalibrationAlm,
                 O_CalibrationWarn => #AD_CalibrationWarn,
                 O_AlarmABCondition => #StopPosAlmCond,
                 H_IAnim => #"H_GBShuttle5Pos2S-MoviFitFCPN".H_2StopPosIAnim[1].H_DWord);
   END_IF;
END_REGION

REGION Network 108: **** 7.3 - Submodule - Machine **** Motor loop MOVIFIT-FC
   // Motor loop MOVIFIT-FC
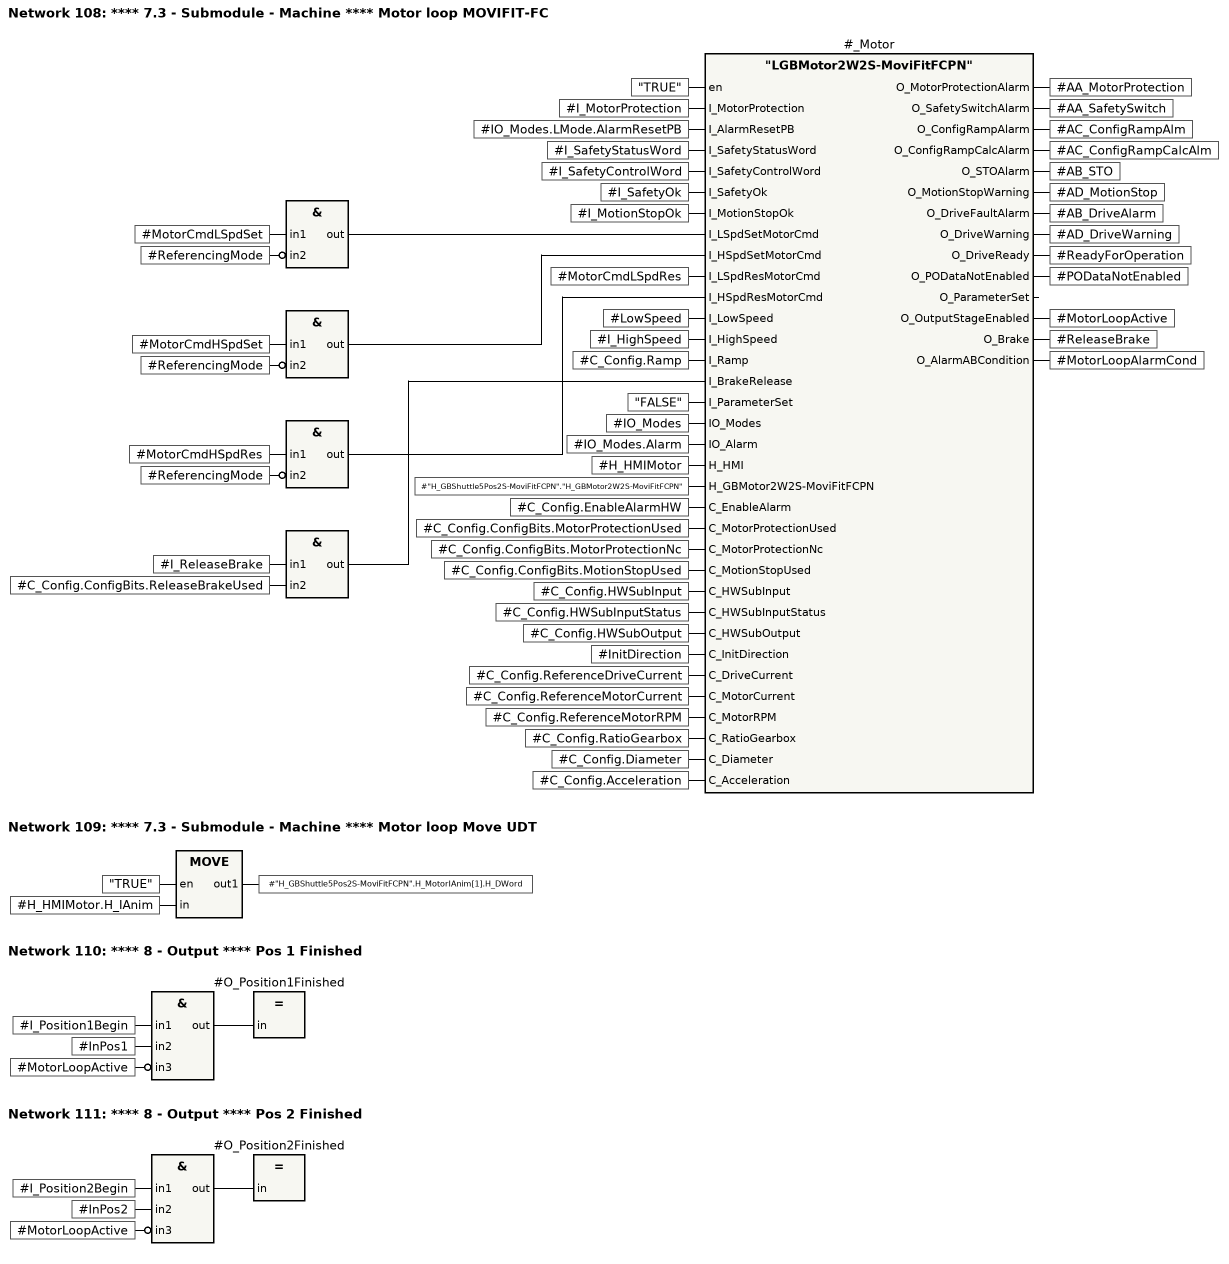
   IF "TRUE" THEN
       #_Motor(I_MotorProtection := #I_MotorProtection,   // "LGBMotor2W2S-MoviFitFCPN"
               I_AlarmResetPB := #IO_Modes.LMode.AlarmResetPB,
               I_SafetyStatusWord := #I_SafetyStatusWord,
               I_SafetyControlWord := #I_SafetyControlWord,
               I_SafetyOk := #I_SafetyOk,
               I_MotionStopOk := #I_MotionStopOk,
               I_LSpdSetMotorCmd := #MotorCmdLSpdSet AND NOT #ReferencingMode,
               I_HSpdSetMotorCmd := #MotorCmdHSpdSet AND NOT #ReferencingMode,
               I_LSpdResMotorCmd := #MotorCmdLSpdRes,
               I_HSpdResMotorCmd := #MotorCmdHSpdRes AND NOT #ReferencingMode,
               I_LowSpeed := #LowSpeed,
               I_HighSpeed := #I_HighSpeed,
               I_Ramp := #C_Config.Ramp,
               I_BrakeRelease := #I_ReleaseBrake AND #C_Config.ConfigBits.ReleaseBrakeUsed,
               I_ParameterSet := "FALSE",
               IO_Modes := #IO_Modes,
               IO_Alarm := #IO_Modes.Alarm,
               H_HMI := #H_HMIMotor,
               "H_GBMotor2W2S-MoviFitFCPN" := #"H_GBShuttle5Pos2S-MoviFitFCPN"."H_GBMotor2W2S-MoviFitFCPN",
               C_EnableAlarm := #C_Config.EnableAlarmHW,
               C_MotorProtectionUsed := #C_Config.ConfigBits.MotorProtectionUsed,
               C_MotorProtectionNc := #C_Config.ConfigBits.MotorProtectionNc,
               C_MotionStopUsed := #C_Config.ConfigBits.MotionStopUsed,
               C_HWSubInput := #C_Config.HWSubInput,
               C_HWSubInputStatus := #C_Config.HWSubInputStatus,
               C_HWSubOutput := #C_Config.HWSubOutput,
               C_InitDirection := #InitDirection,
               C_DriveCurrent := #C_Config.ReferenceDriveCurrent,
               C_MotorCurrent := #C_Config.ReferenceMotorCurrent,
               C_MotorRPM := #C_Config.ReferenceMotorRPM,
               C_RatioGearbox := #C_Config.RatioGearbox,
               C_Diameter := #C_Config.Diameter,
               C_Acceleration := #C_Config.Acceleration,
               O_MotorProtectionAlarm => #AA_MotorProtection,
               O_SafetySwitchAlarm => #AA_SafetySwitch,
               O_ConfigRampAlarm => #AC_ConfigRampAlm,
               O_ConfigRampCalcAlarm => #AC_ConfigRampCalcAlm,
               O_STOAlarm => #AB_STO,
               O_MotionStopWarning => #AD_MotionStop,
               O_DriveFaultAlarm => #AB_DriveAlarm,
               O_DriveWarning => #AD_DriveWarning,
               O_DriveReady => #ReadyForOperation,
               O_PODataNotEnabled => #PODataNotEnabled,
               O_OutputStageEnabled => #MotorLoopActive,
               O_Brake => #ReleaseBrake,
               O_AlarmABCondition => #MotorLoopAlarmCond);
   END_IF;
END_REGION

REGION Network 109: **** 7.3 - Submodule - Machine **** Motor loop Move UDT
   IF "TRUE" THEN #"H_GBShuttle5Pos2S-MoviFitFCPN".H_MotorIAnim[1].H_DWord := #H_HMIMotor.H_IAnim; END_IF;
END_REGION

REGION Network 110: **** 8 - Output **** Pos 1 Finished
   // Pos 1 Finished
   #O_Position1Finished := #I_Position1Begin AND #InPos1 AND NOT #MotorLoopActive;
END_REGION

REGION Network 111: **** 8 - Output **** Pos 2 Finished
   // Pos 1 Finished
   #O_Position2Finished := #I_Position2Begin AND #InPos2 AND NOT #MotorLoopActive;
END_REGION

REGION Network 112: **** 8 - Output **** Pos 3 Finished
   // Pos 3 Finished
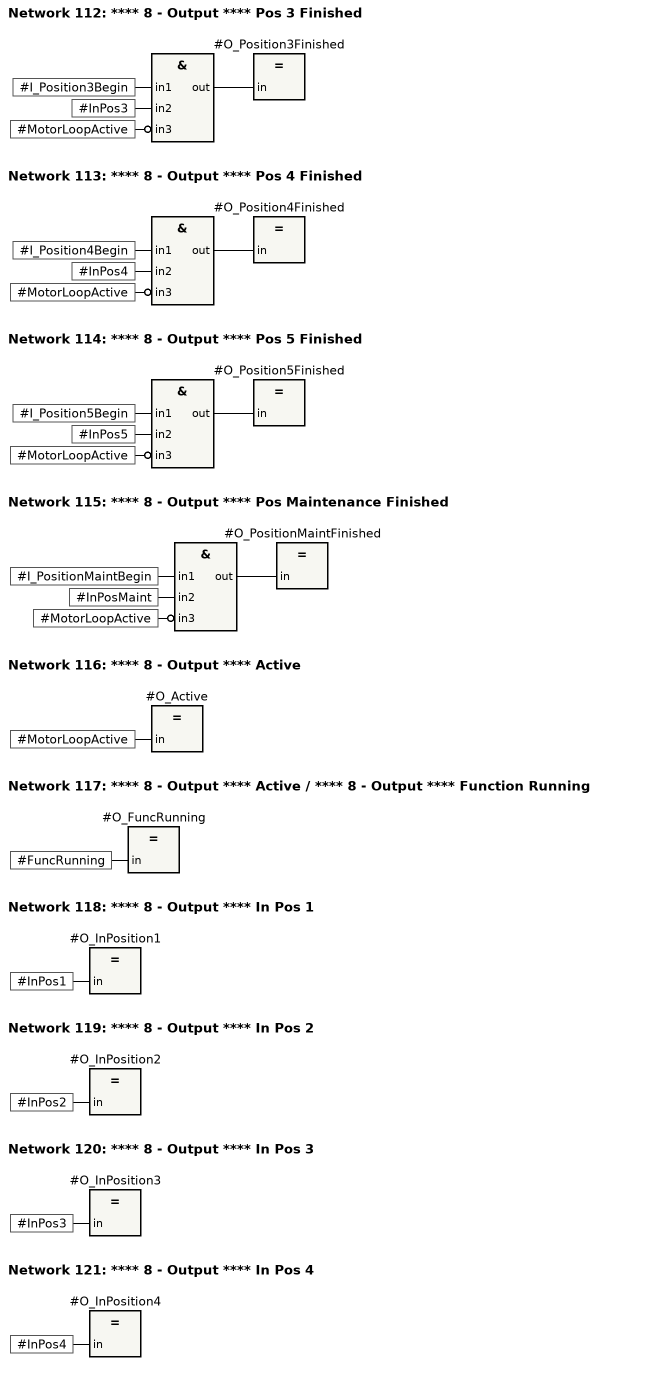
   #O_Position3Finished := #I_Position3Begin AND #InPos3 AND NOT #MotorLoopActive;
END_REGION

REGION Network 113: **** 8 - Output **** Pos 4 Finished
   // Pos 4 Finished
   #O_Position4Finished := #I_Position4Begin AND #InPos4 AND NOT #MotorLoopActive;
END_REGION

REGION Network 114: **** 8 - Output **** Pos 5 Finished
   // Pos 5 Finished
   #O_Position5Finished := #I_Position5Begin AND #InPos5 AND NOT #MotorLoopActive;
END_REGION

REGION Network 115: **** 8 - Output **** Pos Maintenance Finished
   // Pos 4 Finished
   #O_PositionMaintFinished := #I_PositionMaintBegin AND #InPosMaint AND NOT #MotorLoopActive;
END_REGION

REGION Network 116: **** 8 - Output **** Active
   // Active
   #O_Active := #MotorLoopActive;
END_REGION

REGION Network 117: **** 8 - Output **** Active / **** 8 - Output **** Function Running
   // Active
   #O_FuncRunning := #FuncRunning;
END_REGION

REGION Network 118: **** 8 - Output **** In Pos 1
   // In Pos 1
   #O_InPosition1 := #InPos1;
END_REGION

REGION Network 119: **** 8 - Output **** In Pos 2
   // In Pos 2
   #O_InPosition2 := #InPos2;
END_REGION

REGION Network 120: **** 8 - Output **** In Pos 3
   // In Pos 3
   #O_InPosition3 := #InPos3;
END_REGION

REGION Network 121: **** 8 - Output **** In Pos 4
   // In Pos 4
   #O_InPosition4 := #InPos4;
END_REGION

REGION Network 122: **** 8 - Output **** In Pos 5
   // In Pos 5
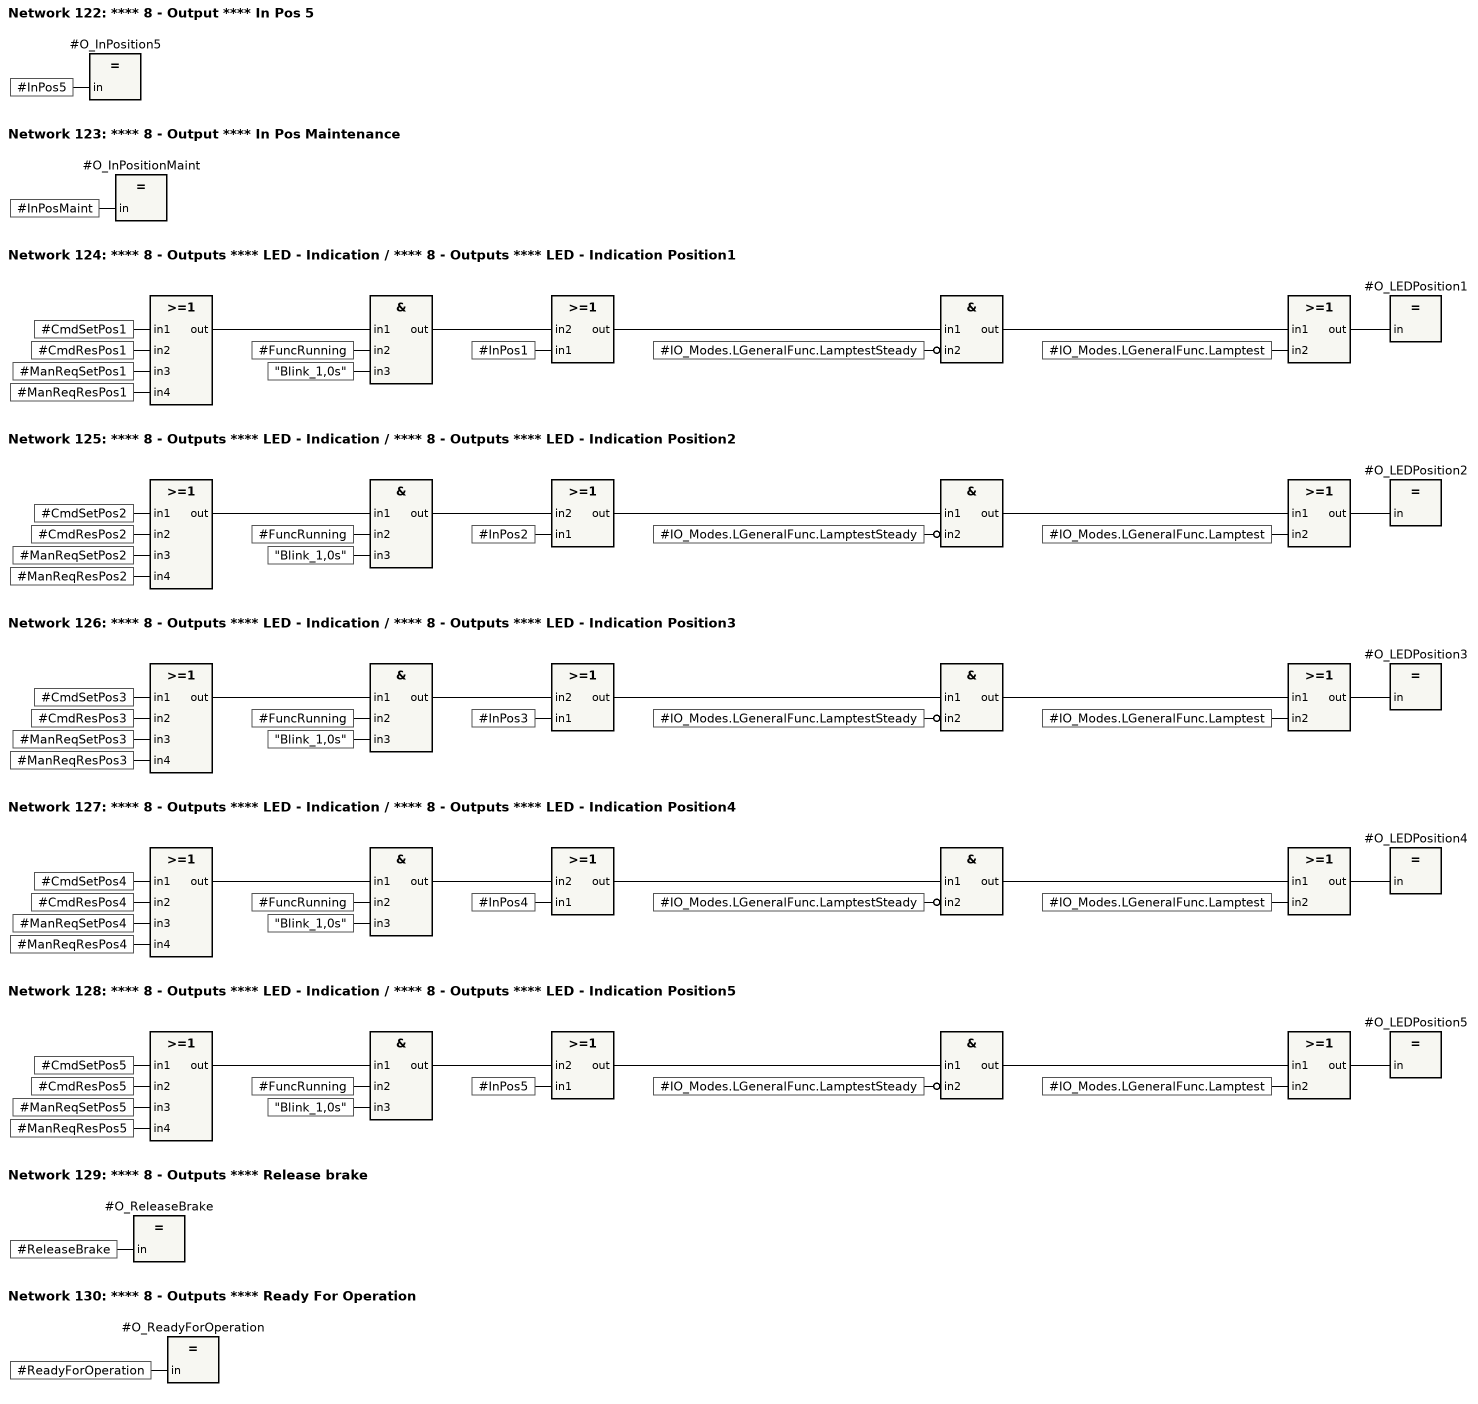
   #O_InPosition5 := #InPos5;
END_REGION

REGION Network 123: **** 8 - Output **** In Pos Maintenance
   // In Pos 4
   #O_InPositionMaint := #InPosMaint;
END_REGION

REGION Network 124: **** 8 - Outputs **** LED - Indication / **** 8 - Outputs **** LED - Indication Position1
   // LED - Indication
   #O_LEDPosition1 := ((((#CmdSetPos1 OR #CmdResPos1 OR #ManReqSetPos1 OR #ManReqResPos1) AND #FuncRunning AND "Blink_1,0s") OR #InPos1) AND NOT #IO_Modes.LGeneralFunc.LamptestSteady) OR #IO_Modes.LGeneralFunc.Lamptest;
END_REGION

REGION Network 125: **** 8 - Outputs **** LED - Indication / **** 8 - Outputs **** LED - Indication Position2
   // LED - Indication
   #O_LEDPosition2 := ((((#CmdSetPos2 OR #CmdResPos2 OR #ManReqSetPos2 OR #ManReqResPos2) AND #FuncRunning AND "Blink_1,0s") OR #InPos2) AND NOT #IO_Modes.LGeneralFunc.LamptestSteady) OR #IO_Modes.LGeneralFunc.Lamptest;
END_REGION

REGION Network 126: **** 8 - Outputs **** LED - Indication / **** 8 - Outputs **** LED - Indication Position3
   // LED - Indication
   #O_LEDPosition3 := ((((#CmdSetPos3 OR #CmdResPos3 OR #ManReqSetPos3 OR #ManReqResPos3) AND #FuncRunning AND "Blink_1,0s") OR #InPos3) AND NOT #IO_Modes.LGeneralFunc.LamptestSteady) OR #IO_Modes.LGeneralFunc.Lamptest;
END_REGION

REGION Network 127: **** 8 - Outputs **** LED - Indication / **** 8 - Outputs **** LED - Indication Position4
   // LED - Indication
   #O_LEDPosition4 := ((((#CmdSetPos4 OR #CmdResPos4 OR #ManReqSetPos4 OR #ManReqResPos4) AND #FuncRunning AND "Blink_1,0s") OR #InPos4) AND NOT #IO_Modes.LGeneralFunc.LamptestSteady) OR #IO_Modes.LGeneralFunc.Lamptest;
END_REGION

REGION Network 128: **** 8 - Outputs **** LED - Indication / **** 8 - Outputs **** LED - Indication Position5
   // LED - Indication
   #O_LEDPosition5 := ((((#CmdSetPos5 OR #CmdResPos5 OR #ManReqSetPos5 OR #ManReqResPos5) AND #FuncRunning AND "Blink_1,0s") OR #InPos5) AND NOT #IO_Modes.LGeneralFunc.LamptestSteady) OR #IO_Modes.LGeneralFunc.Lamptest;
END_REGION

REGION Network 129: **** 8 - Outputs **** Release brake
   // Release brake
   #O_ReleaseBrake := #ReleaseBrake;
END_REGION

REGION Network 130: **** 8 - Outputs **** Ready For Operation
   // Ready For Operation
   #O_ReadyForOperation := #ReadyForOperation;
END_REGION

REGION Network 131: **** 8 - Outputs **** Alarm AB Condition
   // Alarm AB condition
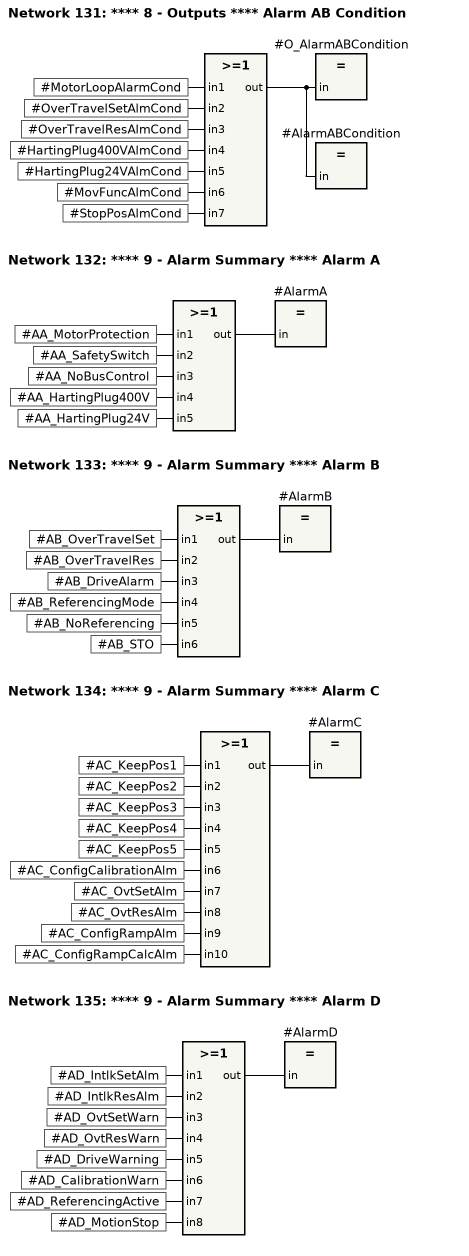
   #O_AlarmABCondition := #MotorLoopAlarmCond OR #OverTravelSetAlmCond OR #OverTravelResAlmCond OR #HartingPlug400VAlmCond OR #HartingPlug24VAlmCond OR #MovFuncAlmCond OR #StopPosAlmCond;
   #AlarmABCondition := #O_AlarmABCondition;
END_REGION

REGION Network 132: **** 9 - Alarm Summary **** Alarm A
   // Alarm A
   #AlarmA := #AA_MotorProtection OR #AA_SafetySwitch OR #AA_NoBusControl OR #AA_HartingPlug400V OR #AA_HartingPlug24V;
END_REGION

REGION Network 133: **** 9 - Alarm Summary **** Alarm B
   // Alarm B
   #AlarmB := #AB_OverTravelSet OR #AB_OverTravelRes OR #AB_DriveAlarm OR #AB_ReferencingMode OR #AB_NoReferencing OR #AB_STO;
END_REGION

REGION Network 134: **** 9 - Alarm Summary **** Alarm C
   // Alarm C
   #AlarmC := #AC_KeepPos1 OR #AC_KeepPos2 OR #AC_KeepPos3 OR #AC_KeepPos4 OR #AC_KeepPos5 OR #AC_ConfigCalibrationAlm OR #AC_OvtSetAlm OR #AC_OvtResAlm OR #AC_ConfigRampAlm OR #AC_ConfigRampCalcAlm;
END_REGION

REGION Network 135: **** 9 - Alarm Summary **** Alarm D
   // Alarm D
   #AlarmD := #AD_IntlkSetAlm OR #AD_IntlkResAlm OR #AD_OvtSetWarn OR #AD_OvtResWarn OR #AD_DriveWarning OR #AD_CalibrationWarn OR #AD_ReferencingActive OR #AD_MotionStop;
END_REGION

REGION Network 136: **** 9 - Alarm Summary **** Alarms To Alarm UDT Alarms To Alarm UDT Get Name
   // Alarms To Alarm UDT Alarms To Alarm UDT Get Name
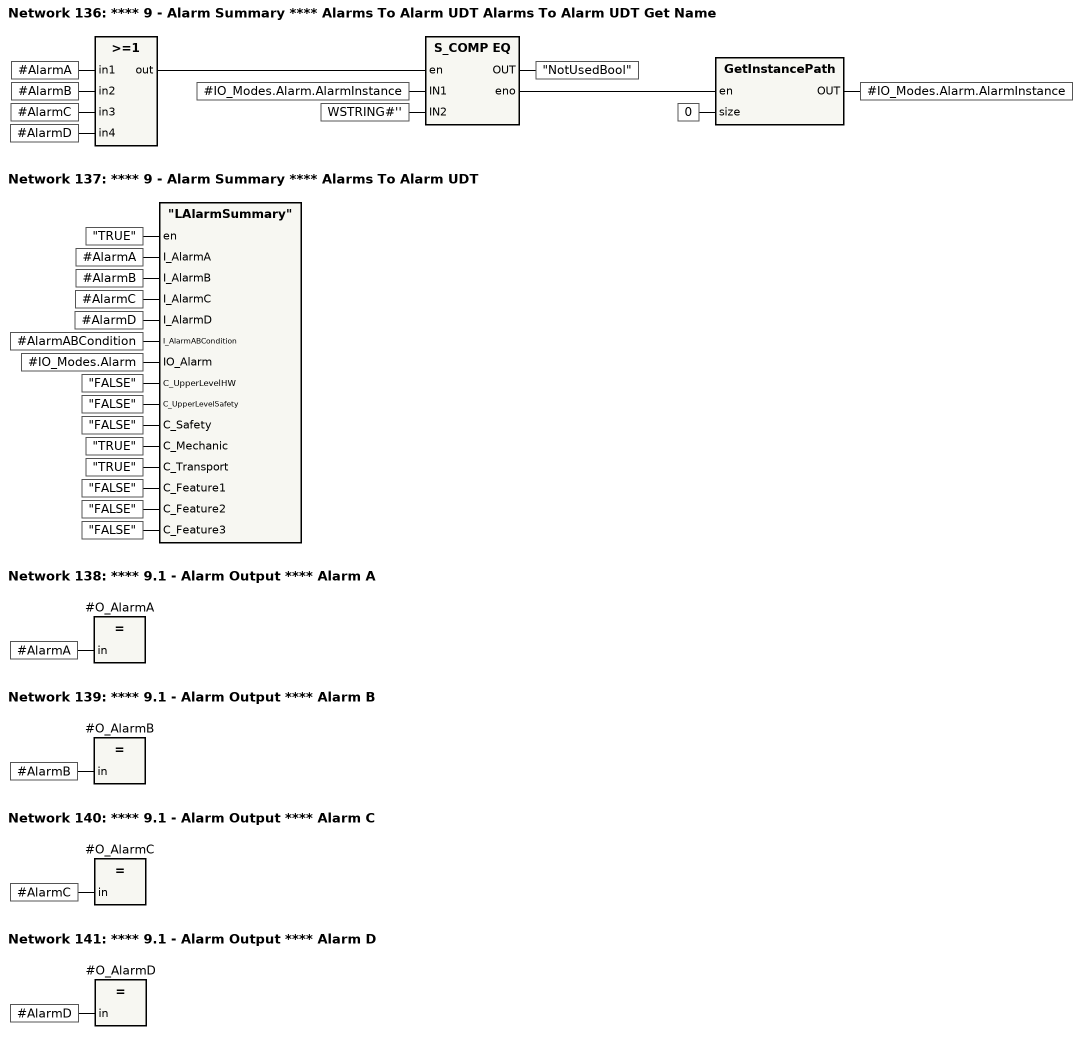
   S_COMP(EN := #AlarmA OR #AlarmB OR #AlarmC OR #AlarmD,
          IN1 := #IO_Modes.Alarm.AlarmInstance,
          IN2 := WSTRING#'',
          OUT => "NotUsedBool",
          ENO => #_w1);
   IF #_w1 THEN GetInstancePath(size := 0, OUT => #IO_Modes.Alarm.AlarmInstance); END_IF;
END_REGION

REGION Network 137: **** 9 - Alarm Summary **** Alarms To Alarm UDT
   // Alarms To Alarm UDT
   IF "TRUE" THEN
       "LAlarmSummary"(I_AlarmA := #AlarmA,
                       I_AlarmB := #AlarmB,
                       I_AlarmC := #AlarmC,
                       I_AlarmD := #AlarmD,
                       I_AlarmABCondition := #AlarmABCondition,
                       IO_Alarm := #IO_Modes.Alarm,
                       C_UpperLevelHW := "FALSE",
                       C_UpperLevelSafety := "FALSE",
                       C_Safety := "FALSE",
                       C_Mechanic := "TRUE",
                       C_Transport := "TRUE",
                       C_Feature1 := "FALSE",
                       C_Feature2 := "FALSE",
                       C_Feature3 := "FALSE");
   END_IF;
END_REGION

REGION Network 138: **** 9.1 - Alarm Output **** Alarm A
   // Alarm A
   #O_AlarmA := #AlarmA;
END_REGION

REGION Network 139: **** 9.1 - Alarm Output **** Alarm B
   // Alarm B
   #O_AlarmB := #AlarmB;
END_REGION

REGION Network 140: **** 9.1 - Alarm Output **** Alarm C
   // Alarm C
   #O_AlarmC := #AlarmC;
END_REGION

REGION Network 141: **** 9.1 - Alarm Output **** Alarm D
   // Alarm D
   #O_AlarmD := #AlarmD;
END_REGION

REGION Network 142: **** 9.2 - Alarm DWord**** Alarm To DWord
   // Alarm To Word
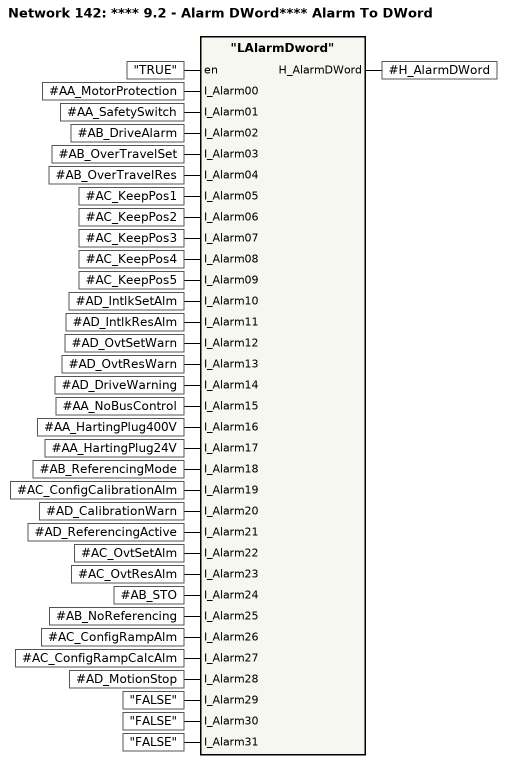
   IF "TRUE" THEN
       "LAlarmDword"(I_Alarm00 := #AA_MotorProtection,
                     I_Alarm01 := #AA_SafetySwitch,
                     I_Alarm02 := #AB_DriveAlarm,
                     I_Alarm03 := #AB_OverTravelSet,
                     I_Alarm04 := #AB_OverTravelRes,
                     I_Alarm05 := #AC_KeepPos1,
                     I_Alarm06 := #AC_KeepPos2,
                     I_Alarm07 := #AC_KeepPos3,
                     I_Alarm08 := #AC_KeepPos4,
                     I_Alarm09 := #AC_KeepPos5,
                     I_Alarm10 := #AD_IntlkSetAlm,
                     I_Alarm11 := #AD_IntlkResAlm,
                     I_Alarm12 := #AD_OvtSetWarn,
                     I_Alarm13 := #AD_OvtResWarn,
                     I_Alarm14 := #AD_DriveWarning,
                     I_Alarm15 := #AA_NoBusControl,
                     I_Alarm16 := #AA_HartingPlug400V,
                     I_Alarm17 := #AA_HartingPlug24V,
                     I_Alarm18 := #AB_ReferencingMode,
                     I_Alarm19 := #AC_ConfigCalibrationAlm,
                     I_Alarm20 := #AD_CalibrationWarn,
                     I_Alarm21 := #AD_ReferencingActive,
                     I_Alarm22 := #AC_OvtSetAlm,
                     I_Alarm23 := #AC_OvtResAlm,
                     I_Alarm24 := #AB_STO,
                     I_Alarm25 := #AB_NoReferencing,
                     I_Alarm26 := #AC_ConfigRampAlm,
                     I_Alarm27 := #AC_ConfigRampCalcAlm,
                     I_Alarm28 := #AD_MotionStop,
                     I_Alarm29 := "FALSE",
                     I_Alarm30 := "FALSE",
                     I_Alarm31 := "FALSE",
                     H_AlarmDWord => #H_AlarmDWord);
   END_IF;
END_REGION
END_FUNCTION_BLOCK
